LIN {X 0,Y 220.383,Z 219.803,A -85,B 0,C 180,E1 -20268.834,E2 -20268.834} C_VEL
LIN {X 0,Y 222.239,Z 208.514,A -85,B 0,C 180,E1 -20275.269,E2 -20275.269} C_VEL
LIN {X 0,Y 223.877,Z 201.722,A -85,B 0,C 180,E1 -20279.111,E2 -20279.111} C_VEL
LIN {X 0,Y 223.579,Z 198.542,A -85,B 0,C 180,E1 -20280.967,E2 -20280.967} C_VEL
LIN {X 0,Y 221.946,Z 190.437,A -85,B 0,C 180,E1 -20285.855,E2 -20285.855} C_VEL
LIN {X 0,Y 220.93,Z 184.96,A -85,B 0,C 180,E1 -20289.374,E2 -20289.374} C_VEL
LIN {X 0,Y 220.782,Z 184.985,A -85,B 0,C 180,E1 -20294.447,E2 -20294.447} C_VEL
LIN {X 0,Y 220.845,Z 184.972,A -85,B 0,C 180,E1 -20298.065,E2 -20298.065} C_VEL
LIN {X 0,Y 220.829,Z 184.976,A -85,B 0,C 180,E1 -20302.71,E2 -20302.71} C_VEL
LIN {X 0,Y 220.813,Z 184.976,A -85,B 0,C 180,E1 -20307.243,E2 -20307.243} C_VEL
LIN {X 0,Y 220.816,Z 184.978,A -85,B 0,C 180,E1 -20311.483,E2 -20311.483} C_VEL
LIN {X 0,Y 220.85,Z 184.972,A -85,B 0,C 180,E1 -20315.563,E2 -20315.563} C_VEL
LIN {X 0,Y 220.873,Z 184.973,A -85,B 0,C 180,E1 -20319.512,E2 -20319.512} C_VEL
LIN {X 0,Y 221.004,Z 184.953,A -85,B 0,C 180,E1 -20323.369,E2 -20323.369} C_VEL
LIN {X 0,Y 221.1,Z 184.943,A -85,B 0,C 180,E1 -20329.005,E2 -20329.005} C_VEL
LIN {X 0,Y 221.276,Z 184.918,A -85,B 0,C 180,E1 -20332.701,E2 -20332.701} C_VEL
LIN {X 0,Y 221.503,Z 184.891,A -85,B 0,C 180,E1 -20338.182,E2 -20338.182} C_VEL
LIN {X 0,Y 221.498,Z 184.891,A -85,B 0,C 180,E1 -20341.818,E2 -20341.818} C_VEL
LIN {X 0,Y 221.277,Z 184.918,A -85,B 0,C 180,E1 -20347.299,E2 -20347.299} C_VEL
LIN {X 0,Y 221.1,Z 184.943,A -85,B 0,C 180,E1 -20350.995,E2 -20350.995} C_VEL
LIN {X 0,Y 221.004,Z 184.953,A -85,B 0,C 180,E1 -20356.631,E2 -20356.631} C_VEL
LIN {X 0,Y 220.876,Z 184.973,A -85,B 0,C 180,E1 -20360.488,E2 -20360.488} C_VEL
LIN {X 0,Y 220.836,Z 184.974,A -85,B 0,C 180,E1 -20364.439,E2 -20364.439} C_VEL
LIN {X 0,Y 220.793,Z 184.981,A -85,B 0,C 180,E1 -20368.52,E2 -20368.52} C_VEL
LIN {X 0,Y 220.807,Z 184.977,A -85,B 0,C 180,E1 -20372.758,E2 -20372.758} C_VEL
LIN {X 0,Y 220.828,Z 184.976,A -85,B 0,C 180,E1 -20377.29,E2 -20377.29} C_VEL
LIN {X 0,Y 220.792,Z 184.979,A -85,B 0,C 180,E1 -20381.947,E2 -20381.947} C_VEL
LIN {X 0,Y 220.768,Z 184.986,A -85,B 0,C 180,E1 -20385.549,E2 -20385.549} C_VEL
LIN {X 0,Y 220.799,Z 184.978,A -85,B 0,C 180,E1 -20390.466,E2 -20390.466} C_VEL
LIN {X 0,Y 220.795,Z 184.983,A -85,B 0,C 180,E1 -20395.048,E2 -20395.048} C_VEL
LIN {X 0,Y 220.863,Z 184.969,A -85,B 0,C 180,E1 -20399.398,E2 -20399.398} C_VEL
LIN {X 0,Y 220.891,Z 184.968,A -85,B 0,C 180,E1 -20403.553,E2 -20403.553} C_VEL
LIN {X 0,Y 220.875,Z 184.968,A -85,B 0,C 180,E1 -20407.556,E2 -20407.556} C_VEL
LIN {X 0,Y 220.982,Z 184.96,A -85,B 0,C 180,E1 -20412.574,E2 -20412.574} C_VEL
LIN {X 0,Y 221.012,Z 184.95,A -85,B 0,C 180,E1 -20417.142,E2 -20417.142} C_VEL
LIN {X 0,Y 221.258,Z 184.923,A -85,B 0,C 180,E1 -20420.865,E2 -20420.865} C_VEL
LIN {X 0,Y 221.312,Z 184.916,A -85,B 0,C 180,E1 -20422.705,E2 -20422.705} C_VEL
LIN {X 0,Y 221.511,Z 184.894,A -85,B 0,C 180,E1 -20428.185,E2 -20428.185} C_VEL
LIN {X 0,Y 221.51,Z 184.894,A -85,B 0,C 180,E1 -20431.821,E2 -20431.821} C_VEL
LIN {X 0,Y 221.314,Z 184.916,A -85,B 0,C 180,E1 -20437.3,E2 -20437.3} C_VEL
LIN {X 0,Y 221.115,Z 184.94,A -85,B 0,C 180,E1 -20440.997,E2 -20440.997} C_VEL
LIN {X 0,Y 221.02,Z 184.952,A -85,B 0,C 180,E1 -20446.632,E2 -20446.632} C_VEL
LIN {X 0,Y 220.886,Z 184.967,A -85,B 0,C 180,E1 -20450.49,E2 -20450.49} C_VEL
LIN {X 0,Y 220.803,Z 184.979,A -85,B 0,C 180,E1 -20454.445,E2 -20454.445} C_VEL
LIN {X 0,Y 220.804,Z 184.979,A -85,B 0,C 180,E1 -20458.521,E2 -20458.521} C_VEL
LIN {X 0,Y 220.818,Z 184.979,A -85,B 0,C 180,E1 -20462.759,E2 -20462.759} C_VEL
LIN {X 0,Y 220.815,Z 184.976,A -85,B 0,C 180,E1 -20467.28,E2 -20467.28} C_VEL
LIN {X 0,Y 220.758,Z 184.985,A -85,B 0,C 180,E1 -20471.959,E2 -20471.959} C_VEL
LIN {X 0,Y 220.776,Z 184.981,A -85,B 0,C 180,E1 -20475.547,E2 -20475.547} C_VEL
LIN {X 0,Y 220.818,Z 184.98,A -85,B 0,C 180,E1 -20480.465,E2 -20480.465} C_VEL
LIN {X 0,Y 221.099,Z 185.049,A -85,B 0,C 180,E1 -20484.682,E2 -20484.682} C_VEL
LIN {X 0,Y 221.776,Z 188.632,A -85,B 0,C 180,E1 -20487.403,E2 -20487.403} C_VEL
LIN {X 0,Y 221.812,Z 191.54,A -85,B 0,C 180,E1 -20489.539,E2 -20489.539} C_VEL
LIN {X 0,Y 220.785,Z 198.517,A -85,B 0,C 180,E1 -20494.55,E2 -20494.55} C_VEL
LIN {X 0,Y 219.989,Z 205.404,A -85,B 0,C 180,E1 -20499.426,E2 -20499.426} C_VEL
LIN {X 0,Y 219.304,Z 213.531,A -85,B 0,C 180,E1 -20505.145,E2 -20505.145} C_VEL
LIN {X 0,Y 219.238,Z 217.231,A -85,B 0,C 180,E1 -20507.739,E2 -20507.739} C_VEL
LIN {X 0,Y 219.799,Z 228.527,A -85,B 0,C 180,E1 -20508.939,E2 -20508.939} C_VEL
LIN {X 0,Y 220.545,Z 237.591,A -85,B 0,C 180,E1 -20510.138,E2 -20510.138} C_VEL
LIN {X 0,Y 220.063,Z 248.605,A -85,B 0,C 180,E1 -20511.998,E2 -20511.998} C_VEL
LIN {X 0,Y 219.533,Z 258.766,A -85,B 0,C 180,E1 -20514.185,E2 -20514.185} C_VEL
LIN {X 0,Y 219.318,Z 266.733,A -85,B 0,C 180,E1 -20516.326,E2 -20516.326} C_VEL
LIN {X 0,Y 218.971,Z 273.609,A -85,B 0,C 180,E1 -20518.621,E2 -20518.621} C_VEL
LIN {X 0,Y 218.926,Z 279.136,A -85,B 0,C 180,E1 -20520.92,E2 -20520.92} C_VEL
LIN {X 0,Y 219.375,Z 284.347,A -85,B 0,C 180,E1 -20523.674,E2 -20523.674} C_VEL
LIN {X 0,Y 220.373,Z 288.134,A -85,B 0,C 180,E1 -20526.409,E2 -20526.409} C_VEL
LIN {X 0,Y 221.649,Z 290.652,A -85,B 0,C 180,E1 -20529.122,E2 -20529.122} C_VEL
LIN {X 0,Y 222.867,Z 291.672,A -85,B 0,C 180,E1 -20530.907,E2 -20530.907} C_VEL
LIN {X 0,Y 224.323,Z 292.16,A -85,B 0,C 180,E1 -20532.669,E2 -20532.669} C_VEL
LIN {X 0,Y 226.248,Z 292.142,A -85,B 0,C 180,E1 -20534.389,E2 -20534.389} C_VEL
LIN {X 0,Y 228.21,Z 291.601,A -85,B 0,C 180,E1 -20536.091,E2 -20536.091} C_VEL
LIN {X 0,Y 230.547,Z 290.562,A -85,B 0,C 180,E1 -20537.749,E2 -20537.749} C_VEL
LIN {X 0,Y 234.632,Z 287.997,A -85,B 0,C 180,E1 -20540.149,E2 -20540.149} C_VEL
LIN {X 0,Y 239.086,Z 284.255,A -85,B 0,C 180,E1 -20542.466,E2 -20542.466} C_VEL
LIN {X 0,Y 242.31,Z 281.065,A -85,B 0,C 180,E1 -20543.958,E2 -20543.958} C_VEL
LIN {X 0,Y 243.63,Z 279.399,A -85,B 0,C 180,E1 -20544.726,E2 -20544.726} C_VEL
LIN {X 0,Y 246.198,Z 274.482,A -85,B 0,C 180,E1 -20547.177,E2 -20547.177} C_VEL
LIN {X 0,Y 248.143,Z 269.374,A -85,B 0,C 180,E1 -20549.712,E2 -20549.712} C_VEL
LIN {X 0,Y 250.03,Z 263.054,A -85,B 0,C 180,E1 -20553.028,E2 -20553.028} C_VEL
LIN {X 0,Y 250.761,Z 259.802,A -85,B 0,C 180,E1 -20555.088,E2 -20555.088} C_VEL
LIN {X 0,Y 250.91,Z 258.67,A -85,B 0,C 180,E1 -20556.03,E2 -20556.03} C_VEL
LIN {X 0,Y 251.075,Z 256.645,A -85,B 0,C 180,E1 -20558.39,E2 -20558.39} C_VEL
LIN {X 0,Y 251.135,Z 255.646,A -85,B 0,C 180,E1 -20560.92,E2 -20560.92} C_VEL
LIN {X 0,Y 251.591,Z 255.794,A -85,B 0,C 180,E1 -20564.296,E2 -20564.296} C_VEL
LIN {X 0,Y 252.211,Z 256.685,A -85,B 0,C 180,E1 -20566.428,E2 -20566.428} C_VEL
LIN {X 0,Y 252.859,Z 258.56,A -85,B 0,C 180,E1 -20568.629,E2 -20568.629} C_VEL
LIN {X 0,Y 253.665,Z 261.185,A -85,B 0,C 180,E1 -20570.875,E2 -20570.875} C_VEL
LIN {X 0,Y 254.443,Z 264.949,A -85,B 0,C 180,E1 -20573.227,E2 -20573.227} C_VEL
LIN {X 0,Y 254.346,Z 266.588,A -85,B 0,C 180,E1 -20573.944,E2 -20573.944} C_VEL
LIN {X 0,Y 251.506,Z 274.816,A -85,B 0,C 180,E1 -20576.501,E2 -20576.501} C_VEL
LIN {X 0,Y 250.329,Z 277.426,A -85,B 0,C 180,E1 -20577.284,E2 -20577.284} C_VEL
LIN {X 0,Y 246.162,Z 283.563,A -85,B 0,C 180,E1 -20578.844,E2 -20578.844} C_VEL
LIN {X 0,Y 243.112,Z 287.073,A -85,B 0,C 180,E1 -20579.71,E2 -20579.71} C_VEL
LIN {X 0,Y 236.799,Z 292.522,A -85,B 0,C 180,E1 -20580.998,E2 -20580.998} C_VEL
LIN {X 0,Y 230.529,Z 297.239,A -85,B 0,C 180,E1 -20582.454,E2 -20582.454} C_VEL
LIN {X 0,Y 227.594,Z 299.611,A -85,B 0,C 180,E1 -20583.576,E2 -20583.576} C_VEL
LIN {X 0,Y 223.623,Z 303.227,A -85,B 0,C 180,E1 -20585.883,E2 -20585.883} C_VEL
LIN {X 0,Y 219.258,Z 306.967,A -85,B 0,C 180,E1 -20589.351,E2 -20589.351} C_VEL
LIN {X 0,Y 215.694,Z 309.301,A -85,B 0,C 180,E1 -20592.945,E2 -20592.945} C_VEL
LIN {X 0,Y 213.363,Z 310.182,A -85,B 0,C 180,E1 -20596.666,E2 -20596.666} C_VEL
LIN {X 0,Y 212.177,Z 309.707,A -85,B 0,C 180,E1 -20600.464,E2 -20600.464} C_VEL
LIN {X 0,Y 212.07,Z 307.767,A -85,B 0,C 180,E1 -20604.291,E2 -20604.291} C_VEL
LIN {X 0,Y 212.215,Z 306.227,A -85,B 0,C 180,E1 -20606.199,E2 -20606.199} C_VEL
LIN {X 0,Y 212.782,Z 303.097,A -85,B 0,C 180,E1 -20609.051,E2 -20609.051} C_VEL
LIN {X 0,Y 213.004,Z 300.337,A -85,B 0,C 180,E1 -20610.942,E2 -20610.942} C_VEL
LIN {X 0,Y 213.038,Z 295.011,A -85,B 0,C 180,E1 -20613.78,E2 -20613.78} C_VEL
LIN {X 0,Y 213.16,Z 288.15,A -85,B 0,C 180,E1 -20616.623,E2 -20616.623} C_VEL
LIN {X 0,Y 213.282,Z 279.264,A -85,B 0,C 180,E1 -20619.48,E2 -20619.48} C_VEL
LIN {X 0,Y 213.737,Z 269.98,A -85,B 0,C 180,E1 -20621.856,E2 -20621.856} C_VEL
LIN {X 0,Y 214.337,Z 259.585,A -85,B 0,C 180,E1 -20623.991,E2 -20623.991} C_VEL
LIN {X 0,Y 215.12,Z 247.855,A -85,B 0,C 180,E1 -20625.876,E2 -20625.876} C_VEL
LIN {X 0,Y 214.061,Z 235.879,A -85,B 0,C 180,E1 -20627.3,E2 -20627.3} C_VEL
LIN {X 0,Y 213.328,Z 223.422,A -85,B 0,C 180,E1 -20628.407,E2 -20628.407} C_VEL
LIN {X 0,Y 213.308,Z 219.864,A -85,B 0,C 180,E1 -20628.683,E2 -20628.683} C_VEL
LIN {X 0,Y 215.064,Z 208.981,A -85,B 0,C 180,E1 -20635.136,E2 -20635.136} C_VEL
LIN {X 0,Y 216.744,Z 202.237,A -85,B 0,C 180,E1 -20639.099,E2 -20639.099} C_VEL
LIN {X 0,Y 216.769,Z 200.445,A -85,B 0,C 180,E1 -20640.164,E2 -20640.164} C_VEL
LIN {X 0,Y 215.08,Z 192.314,A -85,B 0,C 180,E1 -20645.223,E2 -20645.223} C_VEL
LIN {X 0,Y 213.891,Z 185.837,A -85,B 0,C 180,E1 -20649.383,E2 -20649.383} C_VEL
LIN {X 0,Y 213.74,Z 185.859,A -85,B 0,C 180,E1 -20653.665,E2 -20653.665} C_VEL
LIN {X 0,Y 213.804,Z 185.851,A -85,B 0,C 180,E1 -20656.346,E2 -20656.346} C_VEL
LIN {X 0,Y 213.786,Z 185.852,A -85,B 0,C 180,E1 -20659.116,E2 -20659.116} C_VEL
LIN {X 0,Y 213.745,Z 185.859,A -85,B 0,C 180,E1 -20663.712,E2 -20663.712} C_VEL
LIN {X 0,Y 213.76,Z 185.859,A -85,B 0,C 180,E1 -20668.261,E2 -20668.261} C_VEL
LIN {X 0,Y 213.815,Z 185.848,A -85,B 0,C 180,E1 -20672.601,E2 -20672.601} C_VEL
LIN {X 0,Y 213.808,Z 185.85,A -85,B 0,C 180,E1 -20676.972,E2 -20676.972} C_VEL
LIN {X 0,Y 213.932,Z 185.832,A -85,B 0,C 180,E1 -20682.802,E2 -20682.802} C_VEL
LIN {X 0,Y 213.968,Z 185.831,A -85,B 0,C 180,E1 -20686.707,E2 -20686.707} C_VEL
LIN {X 0,Y 214.155,Z 185.805,A -85,B 0,C 180,E1 -20690.556,E2 -20690.556} C_VEL
LIN {X 0,Y 214.214,Z 185.797,A -85,B 0,C 180,E1 -20692.459,E2 -20692.459} C_VEL
LIN {X 0,Y 214.436,Z 185.771,A -85,B 0,C 180,E1 -20698.122,E2 -20698.122} C_VEL
LIN {X 0,Y 214.537,Z 185.756,A -85,B 0,C 180,E1 -20700,E2 -20700} C_VEL
LIN {X 0,Y 214.431,Z 185.772,A -85,B 0,C 180,E1 -20701.878,E2 -20701.878} C_VEL
LIN {X 0,Y 214.215,Z 185.797,A -85,B 0,C 180,E1 -20707.541,E2 -20707.541} C_VEL
LIN {X 0,Y 214.032,Z 185.822,A -85,B 0,C 180,E1 -20711.362,E2 -20711.362} C_VEL
LIN {X 0,Y 213.921,Z 185.835,A -85,B 0,C 180,E1 -20715.238,E2 -20715.238} C_VEL
LIN {X 0,Y 213.825,Z 185.848,A -85,B 0,C 180,E1 -20719.189,E2 -20719.189} C_VEL
LIN {X 0,Y 213.791,Z 185.852,A -85,B 0,C 180,E1 -20723.233,E2 -20723.233} C_VEL
LIN {X 0,Y 213.775,Z 185.853,A -85,B 0,C 180,E1 -20727.43,E2 -20727.43} C_VEL
LIN {X 0,Y 213.75,Z 185.86,A -85,B 0,C 180,E1 -20731.74,E2 -20731.74} C_VEL
LIN {X 0,Y 213.742,Z 185.859,A -85,B 0,C 180,E1 -20736.289,E2 -20736.289} C_VEL
LIN {X 0,Y 213.723,Z 185.861,A -85,B 0,C 180,E1 -20741.123,E2 -20741.123} C_VEL
LIN {X 0,Y 213.739,Z 185.859,A -85,B 0,C 180,E1 -20743.67,E2 -20743.67} C_VEL
LIN {X 0,Y 213.704,Z 185.864,A -85,B 0,C 180,E1 -20748.878,E2 -20748.878} C_VEL
LIN {X 0,Y 213.737,Z 185.86,A -85,B 0,C 180,E1 -20753.715,E2 -20753.715} C_VEL
LIN {X 0,Y 213.789,Z 185.853,A -85,B 0,C 180,E1 -20758.728,E2 -20758.728} C_VEL
LIN {X 0,Y 213.821,Z 185.849,A -85,B 0,C 180,E1 -20762.606,E2 -20762.606} C_VEL
LIN {X 0,Y 213.848,Z 185.845,A -85,B 0,C 180,E1 -20766.956,E2 -20766.956} C_VEL
LIN {X 0,Y 213.93,Z 185.837,A -85,B 0,C 180,E1 -20772.308,E2 -20772.308} C_VEL
LIN {X 0,Y 213.953,Z 185.831,A -85,B 0,C 180,E1 -20776.71,E2 -20776.71} C_VEL
LIN {X 0,Y 214.196,Z 185.804,A -85,B 0,C 180,E1 -20780.561,E2 -20780.561} C_VEL
LIN {X 0,Y 214.248,Z 185.797,A -85,B 0,C 180,E1 -20782.463,E2 -20782.463} C_VEL
LIN {X 0,Y 214.445,Z 185.774,A -85,B 0,C 180,E1 -20788.125,E2 -20788.125} C_VEL
LIN {X 0,Y 214.444,Z 185.774,A -85,B 0,C 180,E1 -20791.881,E2 -20791.881} C_VEL
LIN {X 0,Y 214.251,Z 185.797,A -85,B 0,C 180,E1 -20797.542,E2 -20797.542} C_VEL
LIN {X 0,Y 214.046,Z 185.822,A -85,B 0,C 180,E1 -20801.365,E2 -20801.365} C_VEL
LIN {X 0,Y 213.938,Z 185.835,A -85,B 0,C 180,E1 -20805.239,E2 -20805.239} C_VEL
LIN {X 0,Y 213.838,Z 185.849,A -85,B 0,C 180,E1 -20809.19,E2 -20809.19} C_VEL
LIN {X 0,Y 213.788,Z 185.854,A -85,B 0,C 180,E1 -20813.237,E2 -20813.237} C_VEL
LIN {X 0,Y 213.789,Z 185.853,A -85,B 0,C 180,E1 -20817.429,E2 -20817.429} C_VEL
LIN {X 0,Y 213.764,Z 185.855,A -85,B 0,C 180,E1 -20821.741,E2 -20821.741} C_VEL
LIN {X 0,Y 213.75,Z 185.858,A -85,B 0,C 180,E1 -20826.29,E2 -20826.29} C_VEL
LIN {X 0,Y 213.705,Z 185.864,A -85,B 0,C 180,E1 -20831.13,E2 -20831.13} C_VEL
LIN {X 0,Y 213.709,Z 185.863,A -85,B 0,C 180,E1 -20833.681,E2 -20833.681} C_VEL
LIN {X 0,Y 213.711,Z 185.863,A -85,B 0,C 180,E1 -20836.346,E2 -20836.346} C_VEL
LIN {X 0,Y 213.791,Z 185.853,A -85,B 0,C 180,E1 -20841.348,E2 -20841.348} C_VEL
LIN {X 0,Y 214.063,Z 185.926,A -85,B 0,C 180,E1 -20844.714,E2 -20844.714} C_VEL
LIN {X 0,Y 214.817,Z 190.504,A -85,B 0,C 180,E1 -20848.284,E2 -20848.284} C_VEL
LIN {X 0,Y 214.282,Z 194.938,A -85,B 0,C 180,E1 -20851.583,E2 -20851.583} C_VEL
LIN {X 0,Y 213.301,Z 201.913,A -85,B 0,C 180,E1 -20856.71,E2 -20856.71} C_VEL
LIN {X 0,Y 212.547,Z 208.755,A -85,B 0,C 180,E1 -20861.692,E2 -20861.692} C_VEL
LIN {X 0,Y 212.122,Z 215.525,A -85,B 0,C 180,E1 -20866.59,E2 -20866.59} C_VEL
LIN {X 0,Y 212.156,Z 217.294,A -85,B 0,C 180,E1 -20867.869,E2 -20867.869} C_VEL
LIN {X 0,Y 212.885,Z 229.982,A -85,B 0,C 180,E1 -20869.298,E2 -20869.298} C_VEL
LIN {X 0,Y 213.44,Z 238.744,A -85,B 0,C 180,E1 -20870.524,E2 -20870.524} C_VEL
LIN {X 0,Y 212.968,Z 249.317,A -85,B 0,C 180,E1 -20872.415,E2 -20872.415} C_VEL
LIN {X 0,Y 212.521,Z 257.854,A -85,B 0,C 180,E1 -20874.307,E2 -20874.307} C_VEL
LIN {X 0,Y 212.274,Z 266.55,A -85,B 0,C 180,E1 -20876.679,E2 -20876.679} C_VEL
LIN {X 0,Y 211.927,Z 274.714,A -85,B 0,C 180,E1 -20879.525,E2 -20879.525} C_VEL
LIN {X 0,Y 211.986,Z 280.073,A -85,B 0,C 180,E1 -20881.9,E2 -20881.9} C_VEL
LIN {X 0,Y 212.598,Z 285.136,A -85,B 0,C 180,E1 -20884.741,E2 -20884.741} C_VEL
LIN {X 0,Y 213.806,Z 288.841,A -85,B 0,C 180,E1 -20887.556,E2 -20887.556} C_VEL
LIN {X 0,Y 214.653,Z 290.584,A -85,B 0,C 180,E1 -20889.422,E2 -20889.422} C_VEL
LIN {X 0,Y 215.911,Z 291.844,A -85,B 0,C 180,E1 -20891.263,E2 -20891.263} C_VEL
LIN {X 0,Y 217.433,Z 292.568,A -85,B 0,C 180,E1 -20893.077,E2 -20893.077} C_VEL
LIN {X 0,Y 219.401,Z 292.78,A -85,B 0,C 180,E1 -20894.849,E2 -20894.849} C_VEL
LIN {X 0,Y 221.463,Z 292.511,A -85,B 0,C 180,E1 -20896.595,E2 -20896.595} C_VEL
LIN {X 0,Y 223.875,Z 291.714,A -85,B 0,C 180,E1 -20898.296,E2 -20898.296} C_VEL
LIN {X 0,Y 226.647,Z 290.42,A -85,B 0,C 180,E1 -20899.944,E2 -20899.944} C_VEL
LIN {X 0,Y 231.135,Z 287.501,A -85,B 0,C 180,E1 -20902.339,E2 -20902.339} C_VEL
LIN {X 0,Y 236.095,Z 283.421,A -85,B 0,C 180,E1 -20904.63,E2 -20904.63} C_VEL
LIN {X 0,Y 237.579,Z 281.888,A -85,B 0,C 180,E1 -20905.4,E2 -20905.4} C_VEL
LIN {X 0,Y 240.458,Z 277.435,A -85,B 0,C 180,E1 -20907.882,E2 -20907.882} C_VEL
LIN {X 0,Y 242.733,Z 272.796,A -85,B 0,C 180,E1 -20910.444,E2 -20910.444} C_VEL
LIN {X 0,Y 245.023,Z 267.195,A -85,B 0,C 180,E1 -20913.711,E2 -20913.711} C_VEL
LIN {X 0,Y 246.057,Z 264.079,A -85,B 0,C 180,E1 -20915.974,E2 -20915.974} C_VEL
LIN {X 0,Y 246.476,Z 261.855,A -85,B 0,C 180,E1 -20918.852,E2 -20918.852} C_VEL
LIN {X 0,Y 246.672,Z 261.171,A -85,B 0,C 180,E1 -20920.943,E2 -20920.943} C_VEL
LIN {X 0,Y 246.926,Z 261.137,A -85,B 0,C 180,E1 -20923.086,E2 -20923.086} C_VEL
LIN {X 0,Y 247.401,Z 261.685,A -85,B 0,C 180,E1 -20925.25,E2 -20925.25} C_VEL
LIN {X 0,Y 247.945,Z 263.026,A -85,B 0,C 180,E1 -20927.474,E2 -20927.474} C_VEL
LIN {X 0,Y 248.585,Z 265.172,A -85,B 0,C 180,E1 -20929.76,E2 -20929.76} C_VEL
LIN {X 0,Y 249.153,Z 268.435,A -85,B 0,C 180,E1 -20932.168,E2 -20932.168} C_VEL
LIN {X 0,Y 249.169,Z 270.29,A -85,B 0,C 180,E1 -20933.2,E2 -20933.2} C_VEL
LIN {X 0,Y 246.665,Z 276.32,A -85,B 0,C 180,E1 -20935.258,E2 -20935.258} C_VEL
LIN {X 0,Y 245.111,Z 279.384,A -85,B 0,C 180,E1 -20936.255,E2 -20936.255} C_VEL
LIN {X 0,Y 238.884,Z 287.459,A -85,B 0,C 180,E1 -20938.517,E2 -20938.517} C_VEL
LIN {X 0,Y 232.634,Z 294.496,A -85,B 0,C 180,E1 -20941.092,E2 -20941.092} C_VEL
LIN {X 0,Y 227.594,Z 299.611,A -85,B 0,C 180,E1 -20943.576,E2 -20943.576} C_VEL
LIN {X 0,Y 224.729,Z 301.802,A -85,B 0,C 180,E1 -20944.777,E2 -20944.777} C_VEL
LIN {X 0,Y 218.799,Z 304.886,A -85,B 0,C 180,E1 -20946.677,E2 -20946.677} C_VEL
LIN {X 0,Y 213.226,Z 307.124,A -85,B 0,C 180,E1 -20948.742,E2 -20948.742} C_VEL
LIN {X 0,Y 210.967,Z 308.051,A -85,B 0,C 180,E1 -20950.177,E2 -20950.177} C_VEL
LIN {X 0,Y 208.917,Z 309.041,A -85,B 0,C 180,E1 -20952.373,E2 -20952.373} C_VEL
LIN {X 0,Y 207.468,Z 309.495,A -85,B 0,C 180,E1 -20954.273,E2 -20954.273} C_VEL
LIN {X 0,Y 205.699,Z 309.337,A -85,B 0,C 180,E1 -20958.168,E2 -20958.168} C_VEL
LIN {X 0,Y 205,Z 307.828,A -85,B 0,C 180,E1 -20962.115,E2 -20962.115} C_VEL
LIN {X 0,Y 205.087,Z 306.522,A -85,B 0,C 180,E1 -20964.096,E2 -20964.096} C_VEL
LIN {X 0,Y 205.714,Z 302.691,A -85,B 0,C 180,E1 -20968.039,E2 -20968.039} C_VEL
LIN {X 0,Y 206.06,Z 300.058,A -85,B 0,C 180,E1 -20969.997,E2 -20969.997} C_VEL
LIN {X 0,Y 206.137,Z 294.882,A -85,B 0,C 180,E1 -20972.928,E2 -20972.928} C_VEL
LIN {X 0,Y 206.229,Z 288.195,A -85,B 0,C 180,E1 -20975.865,E2 -20975.865} C_VEL
LIN {X 0,Y 206.274,Z 280.962,A -85,B 0,C 180,E1 -20978.373,E2 -20978.373} C_VEL
LIN {X 0,Y 206.635,Z 272.437,A -85,B 0,C 180,E1 -20980.778,E2 -20980.778} C_VEL
LIN {X 0,Y 207.143,Z 262.818,A -85,B 0,C 180,E1 -20982.986,E2 -20982.986} C_VEL
LIN {X 0,Y 207.862,Z 250.619,A -85,B 0,C 180,E1 -20985.187,E2 -20985.187} C_VEL
LIN {X 0,Y 207.974,Z 245.538,A -85,B 0,C 180,E1 -20985.933,E2 -20985.933} C_VEL
LIN {X 0,Y 206.781,Z 232.916,A -85,B 0,C 180,E1 -20987.404,E2 -20987.404} C_VEL
LIN {X 0,Y 206.262,Z 220.901,A -85,B 0,C 180,E1 -20988.432,E2 -20988.432} C_VEL
LIN {X 0,Y 206.223,Z 219.776,A -85,B 0,C 180,E1 -20988.565,E2 -20988.565} C_VEL
LIN {X 0,Y 208.27,Z 207.727,A -85,B 0,C 180,E1 -20996.016,E2 -20996.016} C_VEL
LIN {X 0,Y 209.665,Z 202.24,A -85,B 0,C 180,E1 -20999.363,E2 -20999.363} C_VEL
LIN {X 0,Y 209.269,Z 199.049,A -85,B 0,C 180,E1 -21001.365,E2 -21001.365} C_VEL
LIN {X 0,Y 207.854,Z 192.27,A -85,B 0,C 180,E1 -21005.757,E2 -21005.757} C_VEL
LIN {X 0,Y 206.826,Z 186.717,A -85,B 0,C 180,E1 -21009.578,E2 -21009.578} C_VEL
LIN {X 0,Y 206.7,Z 186.734,A -85,B 0,C 180,E1 -21015.558,E2 -21015.558} C_VEL
LIN {X 0,Y 206.716,Z 186.734,A -85,B 0,C 180,E1 -21019.761,E2 -21019.761} C_VEL
LIN {X 0,Y 206.716,Z 186.737,A -85,B 0,C 180,E1 -21022.268,E2 -21022.268} C_VEL
LIN {X 0,Y 206.696,Z 186.734,A -85,B 0,C 180,E1 -21027.042,E2 -21027.042} C_VEL
LIN {X 0,Y 206.754,Z 186.73,A -85,B 0,C 180,E1 -21032.096,E2 -21032.096} C_VEL
LIN {X 0,Y 206.743,Z 186.73,A -85,B 0,C 180,E1 -21036.602,E2 -21036.602} C_VEL
LIN {X 0,Y 206.861,Z 186.713,A -85,B 0,C 180,E1 -21042.195,E2 -21042.195} C_VEL
LIN {X 0,Y 206.902,Z 186.711,A -85,B 0,C 180,E1 -21046.245,E2 -21046.245} C_VEL
LIN {X 0,Y 207.093,Z 186.685,A -85,B 0,C 180,E1 -21050.23,E2 -21050.23} C_VEL
LIN {X 0,Y 207.061,Z 186.69,A -85,B 0,C 180,E1 -21054.156,E2 -21054.156} C_VEL
LIN {X 0,Y 207.373,Z 186.651,A -85,B 0,C 180,E1 -21058.058,E2 -21058.058} C_VEL
LIN {X 0,Y 207.502,Z 186.632,A -85,B 0,C 180,E1 -21060,E2 -21060} C_VEL
LIN {X 0,Y 207.368,Z 186.651,A -85,B 0,C 180,E1 -21061.942,E2 -21061.942} C_VEL
LIN {X 0,Y 207.155,Z 186.676,A -85,B 0,C 180,E1 -21067.799,E2 -21067.799} C_VEL
LIN {X 0,Y 206.969,Z 186.702,A -85,B 0,C 180,E1 -21071.756,E2 -21071.756} C_VEL
LIN {X 0,Y 206.855,Z 186.715,A -85,B 0,C 180,E1 -21075.772,E2 -21075.772} C_VEL
LIN {X 0,Y 206.768,Z 186.727,A -85,B 0,C 180,E1 -21079.871,E2 -21079.871} C_VEL
LIN {X 0,Y 206.727,Z 186.734,A -85,B 0,C 180,E1 -21084.077,E2 -21084.077} C_VEL
LIN {X 0,Y 206.677,Z 186.74,A -85,B 0,C 180,E1 -21088.429,E2 -21088.429} C_VEL
LIN {X 0,Y 206.691,Z 186.735,A -85,B 0,C 180,E1 -21092.959,E2 -21092.959} C_VEL
LIN {X 0,Y 206.712,Z 186.732,A -85,B 0,C 180,E1 -21095.322,E2 -21095.322} C_VEL
LIN {X 0,Y 206.665,Z 186.74,A -85,B 0,C 180,E1 -21100.25,E2 -21100.25} C_VEL
LIN {X 0,Y 206.651,Z 186.74,A -85,B 0,C 180,E1 -21104.428,E2 -21104.428} C_VEL
LIN {X 0,Y 206.653,Z 186.741,A -85,B 0,C 180,E1 -21109.752,E2 -21109.752} C_VEL
LIN {X 0,Y 206.692,Z 186.737,A -85,B 0,C 180,E1 -21114.692,E2 -21114.692} C_VEL
LIN {X 0,Y 206.717,Z 186.731,A -85,B 0,C 180,E1 -21119.342,E2 -21119.342} C_VEL
LIN {X 0,Y 206.729,Z 186.732,A -85,B 0,C 180,E1 -21123.775,E2 -21123.775} C_VEL
LIN {X 0,Y 206.754,Z 186.727,A -85,B 0,C 180,E1 -21128.047,E2 -21128.047} C_VEL
LIN {X 0,Y 206.874,Z 186.715,A -85,B 0,C 180,E1 -21132.2,E2 -21132.2} C_VEL
LIN {X 0,Y 206.895,Z 186.712,A -85,B 0,C 180,E1 -21136.248,E2 -21136.248} C_VEL
LIN {X 0,Y 207.132,Z 186.684,A -85,B 0,C 180,E1 -21140.236,E2 -21140.236} C_VEL
LIN {X 0,Y 207.189,Z 186.678,A -85,B 0,C 180,E1 -21142.205,E2 -21142.205} C_VEL
LIN {X 0,Y 207.382,Z 186.653,A -85,B 0,C 180,E1 -21148.061,E2 -21148.061} C_VEL
LIN {X 0,Y 207.484,Z 186.642,A -85,B 0,C 180,E1 -21150.003,E2 -21150.003} C_VEL
LIN {X 0,Y 207.381,Z 186.653,A -85,B 0,C 180,E1 -21151.945,E2 -21151.945} C_VEL
LIN {X 0,Y 207.192,Z 186.678,A -85,B 0,C 180,E1 -21157.801,E2 -21157.801} C_VEL
LIN {X 0,Y 206.979,Z 186.7,A -85,B 0,C 180,E1 -21161.758,E2 -21161.758} C_VEL
LIN {X 0,Y 206.871,Z 186.716,A -85,B 0,C 180,E1 -21165.773,E2 -21165.773} C_VEL
LIN {X 0,Y 206.764,Z 186.726,A -85,B 0,C 180,E1 -21169.874,E2 -21169.874} C_VEL
LIN {X 0,Y 206.705,Z 186.735,A -85,B 0,C 180,E1 -21174.082,E2 -21174.082} C_VEL
LIN {X 0,Y 206.692,Z 186.736,A -85,B 0,C 180,E1 -21178.43,E2 -21178.43} C_VEL
LIN {X 0,Y 206.701,Z 186.739,A -85,B 0,C 180,E1 -21182.96,E2 -21182.96} C_VEL
LIN {X 0,Y 206.679,Z 186.736,A -85,B 0,C 180,E1 -21187.743,E2 -21187.743} C_VEL
LIN {X 0,Y 206.638,Z 186.743,A -85,B 0,C 180,E1 -21191.561,E2 -21191.561} C_VEL
LIN {X 0,Y 206.638,Z 186.742,A -85,B 0,C 180,E1 -21195.584,E2 -21195.584} C_VEL
LIN {X 0,Y 206.684,Z 186.738,A -85,B 0,C 180,E1 -21199.754,E2 -21199.754} C_VEL
LIN {X 0,Y 207.033,Z 186.775,A -85,B 0,C 180,E1 -21204.754,E2 -21204.754} C_VEL
LIN {X 0,Y 207.692,Z 190.556,A -85,B 0,C 180,E1 -21207.78,E2 -21207.78} C_VEL
LIN {X 0,Y 207.404,Z 194.166,A -85,B 0,C 180,E1 -21210.571,E2 -21210.571} C_VEL
LIN {X 0,Y 206.359,Z 201.149,A -85,B 0,C 180,E1 -21215.878,E2 -21215.878} C_VEL
LIN {X 0,Y 205.533,Z 208.004,A -85,B 0,C 180,E1 -21221.044,E2 -21221.044} C_VEL
LIN {X 0,Y 205.051,Z 214.791,A -85,B 0,C 180,E1 -21226.118,E2 -21226.118} C_VEL
LIN {X 0,Y 205.117,Z 217.4,A -85,B 0,C 180,E1 -21228.074,E2 -21228.074} C_VEL
LIN {X 0,Y 205.754,Z 229.252,A -85,B 0,C 180,E1 -21229.421,E2 -21229.421} C_VEL
LIN {X 0,Y 206.395,Z 238.465,A -85,B 0,C 180,E1 -21230.741,E2 -21230.741} C_VEL
LIN {X 0,Y 205.949,Z 248.717,A -85,B 0,C 180,E1 -21232.611,E2 -21232.611} C_VEL
LIN {X 0,Y 205.466,Z 259.399,A -85,B 0,C 180,E1 -21235.095,E2 -21235.095} C_VEL
LIN {X 0,Y 205.234,Z 266.261,A -85,B 0,C 180,E1 -21237.056,E2 -21237.056} C_VEL
LIN {X 0,Y 204.908,Z 274.514,A -85,B 0,C 180,E1 -21240,E2 -21240} C_VEL
LIN {X 0,Y 205.115,Z 280.942,A -85,B 0,C 180,E1 -21242.946,E2 -21242.946} C_VEL
LIN {X 0,Y 205.907,Z 285.873,A -85,B 0,C 180,E1 -21245.877,E2 -21245.877} C_VEL
LIN {X 0,Y 206.795,Z 288.435,A -85,B 0,C 180,E1 -21247.813,E2 -21247.813} C_VEL
LIN {X 0,Y 207.665,Z 290.411,A -85,B 0,C 180,E1 -21249.742,E2 -21249.742} C_VEL
LIN {X 0,Y 208.966,Z 291.882,A -85,B 0,C 180,E1 -21251.642,E2 -21251.642} C_VEL
LIN {X 0,Y 210.557,Z 292.867,A -85,B 0,C 180,E1 -21253.512,E2 -21253.512} C_VEL
LIN {X 0,Y 212.562,Z 293.313,A -85,B 0,C 180,E1 -21255.338,E2 -21255.338} C_VEL
LIN {X 0,Y 214.734,Z 293.3,A -85,B 0,C 180,E1 -21257.131,E2 -21257.131} C_VEL
LIN {X 0,Y 217.224,Z 292.763,A -85,B 0,C 180,E1 -21258.877,E2 -21258.877} C_VEL
LIN {X 0,Y 220.068,Z 291.737,A -85,B 0,C 180,E1 -21260.567,E2 -21260.567} C_VEL
LIN {X 0,Y 224.731,Z 289.268,A -85,B 0,C 180,E1 -21263.011,E2 -21263.011} C_VEL
LIN {X 0,Y 229.88,Z 285.663,A -85,B 0,C 180,E1 -21265.342,E2 -21265.342} C_VEL
LIN {X 0,Y 231.5,Z 284.265,A -85,B 0,C 180,E1 -21266.117,E2 -21266.117} C_VEL
LIN {X 0,Y 233.762,Z 281.58,A -85,B 0,C 180,E1 -21267.775,E2 -21267.775} C_VEL
LIN {X 0,Y 236.699,Z 277.116,A -85,B 0,C 180,E1 -21270.56,E2 -21270.56} C_VEL
LIN {X 0,Y 239.523,Z 271.973,A -85,B 0,C 180,E1 -21273.883,E2 -21273.883} C_VEL
LIN {X 0,Y 240.711,Z 269.524,A -85,B 0,C 180,E1 -21275.728,E2 -21275.728} C_VEL
LIN {X 0,Y 241.395,Z 267.533,A -85,B 0,C 180,E1 -21278.176,E2 -21278.176} C_VEL
LIN {X 0,Y 241.751,Z 266.713,A -85,B 0,C 180,E1 -21279.76,E2 -21279.76} C_VEL
LIN {X 0,Y 241.996,Z 266.365,A -85,B 0,C 180,E1 -21281.91,E2 -21281.91} C_VEL
LIN {X 0,Y 242.361,Z 266.621,A -85,B 0,C 180,E1 -21284.104,E2 -21284.104} C_VEL
LIN {X 0,Y 242.844,Z 267.537,A -85,B 0,C 180,E1 -21286.345,E2 -21286.345} C_VEL
LIN {X 0,Y 243.326,Z 269.307,A -85,B 0,C 180,E1 -21288.674,E2 -21288.674} C_VEL
LIN {X 0,Y 243.775,Z 271.987,A -85,B 0,C 180,E1 -21291.115,E2 -21291.115} C_VEL
LIN {X 0,Y 243.831,Z 273.435,A -85,B 0,C 180,E1 -21292.114,E2 -21292.114} C_VEL
LIN {X 0,Y 243.613,Z 274.527,A -85,B 0,C 180,E1 -21292.709,E2 -21292.709} C_VEL
LIN {X 0,Y 240.366,Z 280.692,A -85,B 0,C 180,E1 -21294.954,E2 -21294.954} C_VEL
LIN {X 0,Y 238.071,Z 283.753,A -85,B 0,C 180,E1 -21295.88,E2 -21295.88} C_VEL
LIN {X 0,Y 232.065,Z 290.386,A -85,B 0,C 180,E1 -21297.992,E2 -21297.992} C_VEL
LIN {X 0,Y 226.551,Z 295.855,A -85,B 0,C 180,E1 -21300.239,E2 -21300.239} C_VEL
LIN {X 0,Y 221.418,Z 300.445,A -85,B 0,C 180,E1 -21302.717,E2 -21302.717} C_VEL
LIN {X 0,Y 217.197,Z 303.792,A -85,B 0,C 180,E1 -21305.121,E2 -21305.121} C_VEL
LIN {X 0,Y 212.623,Z 307.128,A -85,B 0,C 180,E1 -21308.676,E2 -21308.676} C_VEL
LIN {X 0,Y 210.967,Z 308.051,A -85,B 0,C 180,E1 -21310.177,E2 -21310.177} C_VEL
LIN {X 0,Y 208.844,Z 308.8,A -85,B 0,C 180,E1 -21311.669,E2 -21311.669} C_VEL
LIN {X 0,Y 204.087,Z 309.24,A -85,B 0,C 180,E1 -21314.08,E2 -21314.08} C_VEL
LIN {X 0,Y 199.872,Z 308.836,A -85,B 0,C 180,E1 -21316.615,E2 -21316.615} C_VEL
LIN {X 0,Y 198.636,Z 308.28,A -85,B 0,C 180,E1 -21318.263,E2 -21318.263} C_VEL
LIN {X 0,Y 198.07,Z 306.6,A -85,B 0,C 180,E1 -21321.837,E2 -21321.837} C_VEL
LIN {X 0,Y 198.148,Z 305.153,A -85,B 0,C 180,E1 -21323.889,E2 -21323.889} C_VEL
LIN {X 0,Y 198.846,Z 300.988,A -85,B 0,C 180,E1 -21327.971,E2 -21327.971} C_VEL
LIN {X 0,Y 199.182,Z 298.176,A -85,B 0,C 180,E1 -21329.997,E2 -21329.997} C_VEL
LIN {X 0,Y 199.251,Z 292.673,A -85,B 0,C 180,E1 -21333.03,E2 -21333.03} C_VEL
LIN {X 0,Y 199.333,Z 286.875,A -85,B 0,C 180,E1 -21335.561,E2 -21335.561} C_VEL
LIN {X 0,Y 199.364,Z 279.636,A -85,B 0,C 180,E1 -21338.103,E2 -21338.103} C_VEL
LIN {X 0,Y 199.717,Z 270.824,A -85,B 0,C 180,E1 -21340.643,E2 -21340.643} C_VEL
LIN {X 0,Y 200.208,Z 260.923,A -85,B 0,C 180,E1 -21342.928,E2 -21342.928} C_VEL
LIN {X 0,Y 200.848,Z 249.942,A -85,B 0,C 180,E1 -21344.952,E2 -21344.952} C_VEL
LIN {X 0,Y 200.872,Z 244.747,A -85,B 0,C 180,E1 -21345.729,E2 -21345.729} C_VEL
LIN {X 0,Y 199.658,Z 232.007,A -85,B 0,C 180,E1 -21347.252,E2 -21347.252} C_VEL
LIN {X 0,Y 199.185,Z 219.833,A -85,B 0,C 180,E1 -21348.35,E2 -21348.35} C_VEL
LIN {X 0,Y 201.097,Z 208.093,A -85,B 0,C 180,E1 -21355.899,E2 -21355.899} C_VEL
LIN {X 0,Y 202.426,Z 203.099,A -85,B 0,C 180,E1 -21359.078,E2 -21359.078} C_VEL
LIN {X 0,Y 202.45,Z 200.831,A -85,B 0,C 180,E1 -21360.54,E2 -21360.54} C_VEL
LIN {X 0,Y 200.986,Z 193.959,A -85,B 0,C 180,E1 -21365.129,E2 -21365.129} C_VEL
LIN {X 0,Y 199.773,Z 187.595,A -85,B 0,C 180,E1 -21369.667,E2 -21369.667} C_VEL
LIN {X 0,Y 199.638,Z 187.614,A -85,B 0,C 180,E1 -21375.245,E2 -21375.245} C_VEL
LIN {X 0,Y 199.657,Z 187.611,A -85,B 0,C 180,E1 -21378.025,E2 -21378.025} C_VEL
LIN {X 0,Y 199.671,Z 187.613,A -85,B 0,C 180,E1 -21380.74,E2 -21380.74} C_VEL
LIN {X 0,Y 199.624,Z 187.615,A -85,B 0,C 180,E1 -21385.715,E2 -21385.715} C_VEL
LIN {X 0,Y 199.686,Z 187.612,A -85,B 0,C 180,E1 -21388.134,E2 -21388.134} C_VEL
LIN {X 0,Y 199.674,Z 187.609,A -85,B 0,C 180,E1 -21392.77,E2 -21392.77} C_VEL
LIN {X 0,Y 199.703,Z 187.608,A -85,B 0,C 180,E1 -21397.225,E2 -21397.225} C_VEL
LIN {X 0,Y 199.784,Z 187.596,A -85,B 0,C 180,E1 -21401.757,E2 -21401.757} C_VEL
LIN {X 0,Y 199.836,Z 187.593,A -85,B 0,C 180,E1 -21405.748,E2 -21405.748} C_VEL
LIN {X 0,Y 200.058,Z 187.562,A -85,B 0,C 180,E1 -21409.883,E2 -21409.883} C_VEL
LIN {X 0,Y 200.023,Z 187.567,A -85,B 0,C 180,E1 -21413.949,E2 -21413.949} C_VEL
LIN {X 0,Y 200.312,Z 187.53,A -85,B 0,C 180,E1 -21417.989,E2 -21417.989} C_VEL
LIN {X 0,Y 200.466,Z 187.508,A -85,B 0,C 180,E1 -21420,E2 -21420} C_VEL
LIN {X 0,Y 200.015,Z 187.569,A -85,B 0,C 180,E1 -21424.03,E2 -21424.03} C_VEL
LIN {X 0,Y 200.099,Z 187.556,A -85,B 0,C 180,E1 -21428.076,E2 -21428.076} C_VEL
LIN {X 0,Y 199.901,Z 187.584,A -85,B 0,C 180,E1 -21432.178,E2 -21432.178} C_VEL
LIN {X 0,Y 199.792,Z 187.596,A -85,B 0,C 180,E1 -21436.344,E2 -21436.344} C_VEL
LIN {X 0,Y 199.679,Z 187.612,A -85,B 0,C 180,E1 -21440.607,E2 -21440.607} C_VEL
LIN {X 0,Y 199.639,Z 187.612,A -85,B 0,C 180,E1 -21444.989,E2 -21444.989} C_VEL
LIN {X 0,Y 199.597,Z 187.621,A -85,B 0,C 180,E1 -21449.535,E2 -21449.535} C_VEL
LIN {X 0,Y 199.64,Z 187.614,A -85,B 0,C 180,E1 -21452.348,E2 -21452.348} C_VEL
LIN {X 0,Y 199.63,Z 187.616,A -85,B 0,C 180,E1 -21456.762,E2 -21456.762} C_VEL
LIN {X 0,Y 199.631,Z 187.618,A -85,B 0,C 180,E1 -21459.323,E2 -21459.323} C_VEL
LIN {X 0,Y 199.591,Z 187.618,A -85,B 0,C 180,E1 -21462.321,E2 -21462.321} C_VEL
LIN {X 0,Y 199.586,Z 187.622,A -85,B 0,C 180,E1 -21465.236,E2 -21465.236} C_VEL
LIN {X 0,Y 199.572,Z 187.624,A -85,B 0,C 180,E1 -21468.008,E2 -21468.008} C_VEL
LIN {X 0,Y 199.603,Z 187.618,A -85,B 0,C 180,E1 -21470.77,E2 -21470.77} C_VEL
LIN {X 0,Y 199.607,Z 187.62,A -85,B 0,C 180,E1 -21475.717,E2 -21475.717} C_VEL
LIN {X 0,Y 199.695,Z 187.607,A -85,B 0,C 180,E1 -21478.14,E2 -21478.14} C_VEL
LIN {X 0,Y 199.683,Z 187.611,A -85,B 0,C 180,E1 -21482.775,E2 -21482.775} C_VEL
LIN {X 0,Y 199.735,Z 187.602,A -85,B 0,C 180,E1 -21487.232,E2 -21487.232} C_VEL
LIN {X 0,Y 199.835,Z 187.591,A -85,B 0,C 180,E1 -21491.725,E2 -21491.725} C_VEL
LIN {X 0,Y 199.835,Z 187.59,A -85,B 0,C 180,E1 -21495.752,E2 -21495.752} C_VEL
LIN {X 0,Y 200.075,Z 187.561,A -85,B 0,C 180,E1 -21499.888,E2 -21499.888} C_VEL
LIN {X 0,Y 200.132,Z 187.556,A -85,B 0,C 180,E1 -21501.928,E2 -21501.928} C_VEL
LIN {X 0,Y 200.322,Z 187.531,A -85,B 0,C 180,E1 -21507.993,E2 -21507.993} C_VEL
LIN {X 0,Y 200.452,Z 187.518,A -85,B 0,C 180,E1 -21510.003,E2 -21510.003} C_VEL
LIN {X 0,Y 200.321,Z 187.532,A -85,B 0,C 180,E1 -21512.014,E2 -21512.014} C_VEL
LIN {X 0,Y 200.135,Z 187.555,A -85,B 0,C 180,E1 -21518.078,E2 -21518.078} C_VEL
LIN {X 0,Y 199.91,Z 187.578,A -85,B 0,C 180,E1 -21522.18,E2 -21522.18} C_VEL
LIN {X 0,Y 199.809,Z 187.594,A -85,B 0,C 180,E1 -21526.346,E2 -21526.346} C_VEL
LIN {X 0,Y 199.68,Z 187.608,A -85,B 0,C 180,E1 -21530.611,E2 -21530.611} C_VEL
LIN {X 0,Y 199.63,Z 187.619,A -85,B 0,C 180,E1 -21534.993,E2 -21534.993} C_VEL
LIN {X 0,Y 199.612,Z 187.615,A -85,B 0,C 180,E1 -21539.536,E2 -21539.536} C_VEL
LIN {X 0,Y 199.671,Z 187.611,A -85,B 0,C 180,E1 -21542.355,E2 -21542.355} C_VEL
LIN {X 0,Y 199.626,Z 187.618,A -85,B 0,C 180,E1 -21546.766,E2 -21546.766} C_VEL
LIN {X 0,Y 199.602,Z 187.618,A -85,B 0,C 180,E1 -21549.333,E2 -21549.333} C_VEL
LIN {X 0,Y 199.573,Z 187.625,A -85,B 0,C 180,E1 -21552.31,E2 -21552.31} C_VEL
LIN {X 0,Y 199.584,Z 187.621,A -85,B 0,C 180,E1 -21555.23,E2 -21555.23} C_VEL
LIN {X 0,Y 199.682,Z 187.611,A -85,B 0,C 180,E1 -21560.747,E2 -21560.747} C_VEL
LIN {X 0,Y 199.989,Z 187.69,A -85,B 0,C 180,E1 -21564.869,E2 -21564.869} C_VEL
LIN {X 0,Y 200.592,Z 190.541,A -85,B 0,C 180,E1 -21567.237,E2 -21567.237} C_VEL
LIN {X 0,Y 200.557,Z 193.314,A -85,B 0,C 180,E1 -21569.462,E2 -21569.462} C_VEL
LIN {X 0,Y 199.598,Z 198.947,A -85,B 0,C 180,E1 -21573.888,E2 -21573.888} C_VEL
LIN {X 0,Y 198.861,Z 204.494,A -85,B 0,C 180,E1 -21578.218,E2 -21578.218} C_VEL
LIN {X 0,Y 198.145,Z 211.299,A -85,B 0,C 180,E1 -21583.516,E2 -21583.516} C_VEL
LIN {X 0,Y 198.063,Z 217.492,A -85,B 0,C 180,E1 -21588.292,E2 -21588.292} C_VEL
LIN {X 0,Y 198.624,Z 228.33,A -85,B 0,C 180,E1 -21589.552,E2 -21589.552} C_VEL
LIN {X 0,Y 199.374,Z 236.807,A -85,B 0,C 180,E1 -21590.771,E2 -21590.771} C_VEL
LIN {X 0,Y 198.945,Z 247.55,A -85,B 0,C 180,E1 -21592.743,E2 -21592.743} C_VEL
LIN {X 0,Y 198.502,Z 256.996,A -85,B 0,C 180,E1 -21594.922,E2 -21594.922} C_VEL
LIN {X 0,Y 198.303,Z 264.264,A -85,B 0,C 180,E1 -21596.953,E2 -21596.953} C_VEL
LIN {X 0,Y 197.965,Z 271.659,A -85,B 0,C 180,E1 -21599.492,E2 -21599.492} C_VEL
LIN {X 0,Y 198.024,Z 278.78,A -85,B 0,C 180,E1 -21602.543,E2 -21602.543} C_VEL
LIN {X 0,Y 198.543,Z 283.492,A -85,B 0,C 180,E1 -21605.077,E2 -21605.077} C_VEL
LIN {X 0,Y 199.79,Z 287.878,A -85,B 0,C 180,E1 -21608.089,E2 -21608.089} C_VEL
LIN {X 0,Y 200.687,Z 290.111,A -85,B 0,C 180,E1 -21610.085,E2 -21610.085} C_VEL
LIN {X 0,Y 202.033,Z 291.8,A -85,B 0,C 180,E1 -21612.047,E2 -21612.047} C_VEL
LIN {X 0,Y 203.673,Z 293.019,A -85,B 0,C 180,E1 -21613.978,E2 -21613.978} C_VEL
LIN {X 0,Y 205.743,Z 293.73,A -85,B 0,C 180,E1 -21615.859,E2 -21615.859} C_VEL
LIN {X 0,Y 207.986,Z 293.955,A -85,B 0,C 180,E1 -21617.705,E2 -21617.705} C_VEL
LIN {X 0,Y 210.577,Z 293.701,A -85,B 0,C 180,E1 -21619.497,E2 -21619.497} C_VEL
LIN {X 0,Y 213.502,Z 292.939,A -85,B 0,C 180,E1 -21621.229,E2 -21621.229} C_VEL
LIN {X 0,Y 216.704,Z 291.714,A -85,B 0,C 180,E1 -21622.903,E2 -21622.903} C_VEL
LIN {X 0,Y 221.833,Z 288.939,A -85,B 0,C 180,E1 -21625.322,E2 -21625.322} C_VEL
LIN {X 0,Y 225.419,Z 286.526,A -85,B 0,C 180,E1 -21626.877,E2 -21626.877} C_VEL
LIN {X 0,Y 227.901,Z 284.125,A -85,B 0,C 180,E1 -21628.554,E2 -21628.554} C_VEL
LIN {X 0,Y 231.593,Z 279.538,A -85,B 0,C 180,E1 -21631.817,E2 -21631.817} C_VEL
LIN {X 0,Y 234.342,Z 275.567,A -85,B 0,C 180,E1 -21634.738,E2 -21634.738} C_VEL
LIN {X 0,Y 235.569,Z 273.545,A -85,B 0,C 180,E1 -21636.633,E2 -21636.633} C_VEL
LIN {X 0,Y 236.483,Z 271.848,A -85,B 0,C 180,E1 -21639.401,E2 -21639.401} C_VEL
LIN {X 0,Y 236.786,Z 271.451,A -85,B 0,C 180,E1 -21640.767,E2 -21640.767} C_VEL
LIN {X 0,Y 237.116,Z 271.445,A -85,B 0,C 180,E1 -21642.978,E2 -21642.978} C_VEL
LIN {X 0,Y 237.525,Z 272.048,A -85,B 0,C 180,E1 -21645.245,E2 -21645.245} C_VEL
LIN {X 0,Y 237.917,Z 273.381,A -85,B 0,C 180,E1 -21647.604,E2 -21647.604} C_VEL
LIN {X 0,Y 238.317,Z 275.53,A -85,B 0,C 180,E1 -21650.063,E2 -21650.063} C_VEL
LIN {X 0,Y 238.287,Z 277.59,A -85,B 0,C 180,E1 -21651.727,E2 -21651.727} C_VEL
LIN {X 0,Y 236.655,Z 280.597,A -85,B 0,C 180,E1 -21653.029,E2 -21653.029} C_VEL
LIN {X 0,Y 234.865,Z 283.265,A -85,B 0,C 180,E1 -21654.054,E2 -21654.054} C_VEL
LIN {X 0,Y 228.212,Z 290.214,A -85,B 0,C 180,E1 -21656.333,E2 -21656.333} C_VEL
LIN {X 0,Y 222.553,Z 295.401,A -85,B 0,C 180,E1 -21658.488,E2 -21658.488} C_VEL
LIN {X 0,Y 217.041,Z 299.914,A -85,B 0,C 180,E1 -21660.938,E2 -21660.938} C_VEL
LIN {X 0,Y 213.771,Z 302.312,A -85,B 0,C 180,E1 -21662.593,E2 -21662.593} C_VEL
LIN {X 0,Y 210.792,Z 304.284,A -85,B 0,C 180,E1 -21664.312,E2 -21664.312} C_VEL
LIN {X 0,Y 206.025,Z 307.19,A -85,B 0,C 180,E1 -21667.958,E2 -21667.958} C_VEL
LIN {X 0,Y 202.163,Z 308.7,A -85,B 0,C 180,E1 -21671.764,E2 -21671.764} C_VEL
LIN {X 0,Y 199.568,Z 308.882,A -85,B 0,C 180,E1 -21675.726,E2 -21675.726} C_VEL
LIN {X 0,Y 198.636,Z 308.28,A -85,B 0,C 180,E1 -21678.263,E2 -21678.263} C_VEL
LIN {X 0,Y 197.604,Z 307.537,A -85,B 0,C 180,E1 -21679.929,E2 -21679.929} C_VEL
LIN {X 0,Y 194.562,Z 305.306,A -85,B 0,C 180,E1 -21682.612,E2 -21682.612} C_VEL
LIN {X 0,Y 192.342,Z 302.912,A -85,B 0,C 180,E1 -21684.776,E2 -21684.776} C_VEL
LIN {X 0,Y 191.646,Z 300.911,A -85,B 0,C 180,E1 -21686.439,E2 -21686.439} C_VEL
LIN {X 0,Y 191.713,Z 300.239,A -85,B 0,C 180,E1 -21686.998,E2 -21686.998} C_VEL
LIN {X 0,Y 192.205,Z 297.736,A -85,B 0,C 180,E1 -21688.949,E2 -21688.949} C_VEL
LIN {X 0,Y 192.378,Z 294.348,A -85,B 0,C 180,E1 -21691.043,E2 -21691.043} C_VEL
LIN {X 0,Y 192.462,Z 287.976,A -85,B 0,C 180,E1 -21694.185,E2 -21694.185} C_VEL
LIN {X 0,Y 192.502,Z 281.232,A -85,B 0,C 180,E1 -21696.811,E2 -21696.811} C_VEL
LIN {X 0,Y 192.717,Z 271.948,A -85,B 0,C 180,E1 -21699.709,E2 -21699.709} C_VEL
LIN {X 0,Y 193.157,Z 262.584,A -85,B 0,C 180,E1 -21702.073,E2 -21702.073} C_VEL
LIN {X 0,Y 193.775,Z 250.63,A -85,B 0,C 180,E1 -21704.435,E2 -21704.435} C_VEL
LIN {X 0,Y 193.893,Z 244.805,A -85,B 0,C 180,E1 -21705.367,E2 -21705.367} C_VEL
LIN {X 0,Y 192.632,Z 231.999,A -85,B 0,C 180,E1 -21706.966,E2 -21706.966} C_VEL
LIN {X 0,Y 192.142,Z 219.834,A -85,B 0,C 180,E1 -21708.1,E2 -21708.1} C_VEL
LIN {X 0,Y 194.329,Z 206.787,A -85,B 0,C 180,E1 -21716.872,E2 -21716.872} C_VEL
LIN {X 0,Y 195.273,Z 203.484,A -85,B 0,C 180,E1 -21719.066,E2 -21719.066} C_VEL
LIN {X 0,Y 195.421,Z 201.588,A -85,B 0,C 180,E1 -21720.33,E2 -21720.33} C_VEL
LIN {X 0,Y 193.84,Z 194.2,A -85,B 0,C 180,E1 -21725.454,E2 -21725.454} C_VEL
LIN {X 0,Y 192.742,Z 188.471,A -85,B 0,C 180,E1 -21729.585,E2 -21729.585} C_VEL
LIN {X 0,Y 192.585,Z 188.494,A -85,B 0,C 180,E1 -21736.103,E2 -21736.103} C_VEL
LIN {X 0,Y 192.582,Z 188.495,A -85,B 0,C 180,E1 -21740.023,E2 -21740.023} C_VEL
LIN {X 0,Y 192.592,Z 188.493,A -85,B 0,C 180,E1 -21744.277,E2 -21744.277} C_VEL
LIN {X 0,Y 192.589,Z 188.494,A -85,B 0,C 180,E1 -21749.277,E2 -21749.277} C_VEL
LIN {X 0,Y 192.65,Z 188.488,A -85,B 0,C 180,E1 -21751.689,E2 -21751.689} C_VEL
LIN {X 0,Y 192.674,Z 188.483,A -85,B 0,C 180,E1 -21756.344,E2 -21756.344} C_VEL
LIN {X 0,Y 192.72,Z 188.478,A -85,B 0,C 180,E1 -21761.457,E2 -21761.457} C_VEL
LIN {X 0,Y 192.76,Z 188.473,A -85,B 0,C 180,E1 -21765.213,E2 -21765.213} C_VEL
LIN {X 0,Y 192.969,Z 188.446,A -85,B 0,C 180,E1 -21769.508,E2 -21769.508} C_VEL
LIN {X 0,Y 193.049,Z 188.435,A -85,B 0,C 180,E1 -21771.627,E2 -21771.627} C_VEL
LIN {X 0,Y 193.254,Z 188.41,A -85,B 0,C 180,E1 -21777.916,E2 -21777.916} C_VEL
LIN {X 0,Y 193.43,Z 188.384,A -85,B 0,C 180,E1 -21780,E2 -21780} C_VEL
LIN {X 0,Y 192.962,Z 188.448,A -85,B 0,C 180,E1 -21784.177,E2 -21784.177} C_VEL
LIN {X 0,Y 193.049,Z 188.435,A -85,B 0,C 180,E1 -21788.373,E2 -21788.373} C_VEL
LIN {X 0,Y 192.841,Z 188.465,A -85,B 0,C 180,E1 -21792.631,E2 -21792.631} C_VEL
LIN {X 0,Y 192.746,Z 188.471,A -85,B 0,C 180,E1 -21796.96,E2 -21796.96} C_VEL
LIN {X 0,Y 192.609,Z 188.491,A -85,B 0,C 180,E1 -21801.4,E2 -21801.4} C_VEL
LIN {X 0,Y 192.628,Z 188.489,A -85,B 0,C 180,E1 -21804.21,E2 -21804.21} C_VEL
LIN {X 0,Y 192.591,Z 188.494,A -85,B 0,C 180,E1 -21808.868,E2 -21808.868} C_VEL
LIN {X 0,Y 192.585,Z 188.492,A -85,B 0,C 180,E1 -21813.188,E2 -21813.188} C_VEL
LIN {X 0,Y 192.6,Z 188.492,A -85,B 0,C 180,E1 -21816.61,E2 -21816.61} C_VEL
LIN {X 0,Y 192.527,Z 188.501,A -85,B 0,C 180,E1 -21821.077,E2 -21821.077} C_VEL
LIN {X 0,Y 192.513,Z 188.504,A -85,B 0,C 180,E1 -21826.087,E2 -21826.087} C_VEL
LIN {X 0,Y 192.511,Z 188.501,A -85,B 0,C 180,E1 -21830.054,E2 -21830.054} C_VEL
LIN {X 0,Y 192.554,Z 188.498,A -85,B 0,C 180,E1 -21834.273,E2 -21834.273} C_VEL
LIN {X 0,Y 192.604,Z 188.494,A -85,B 0,C 180,E1 -21837.061,E2 -21837.061} C_VEL
LIN {X 0,Y 192.66,Z 188.484,A -85,B 0,C 180,E1 -21841.695,E2 -21841.695} C_VEL
LIN {X 0,Y 192.702,Z 188.48,A -85,B 0,C 180,E1 -21846.352,E2 -21846.352} C_VEL
LIN {X 0,Y 192.779,Z 188.47,A -85,B 0,C 180,E1 -21851.417,E2 -21851.417} C_VEL
LIN {X 0,Y 192.821,Z 188.461,A -85,B 0,C 180,E1 -21857.371,E2 -21857.371} C_VEL
LIN {X 0,Y 193.019,Z 188.439,A -85,B 0,C 180,E1 -21859.514,E2 -21859.514} C_VEL
LIN {X 0,Y 193.005,Z 188.442,A -85,B 0,C 180,E1 -21863.732,E2 -21863.732} C_VEL
LIN {X 0,Y 193.264,Z 188.41,A -85,B 0,C 180,E1 -21867.919,E2 -21867.919} C_VEL
LIN {X 0,Y 193.42,Z 188.394,A -85,B 0,C 180,E1 -21870.003,E2 -21870.003} C_VEL
LIN {X 0,Y 192.977,Z 188.443,A -85,B 0,C 180,E1 -21874.18,E2 -21874.18} C_VEL
LIN {X 0,Y 193.082,Z 188.433,A -85,B 0,C 180,E1 -21878.375,E2 -21878.375} C_VEL
LIN {X 0,Y 193.013,Z 188.44,A -85,B 0,C 180,E1 -21880.541,E2 -21880.541} C_VEL
LIN {X 0,Y 192.761,Z 188.473,A -85,B 0,C 180,E1 -21886.962,E2 -21886.962} C_VEL
LIN {X 0,Y 192.602,Z 188.49,A -85,B 0,C 180,E1 -21891.405,E2 -21891.405} C_VEL
LIN {X 0,Y 192.624,Z 188.489,A -85,B 0,C 180,E1 -21894.197,E2 -21894.197} C_VEL
LIN {X 0,Y 192.605,Z 188.492,A -85,B 0,C 180,E1 -21898.868,E2 -21898.868} C_VEL
LIN {X 0,Y 192.6,Z 188.494,A -85,B 0,C 180,E1 -21903.189,E2 -21903.189} C_VEL
LIN {X 0,Y 192.549,Z 188.497,A -85,B 0,C 180,E1 -21908.356,E2 -21908.356} C_VEL
LIN {X 0,Y 192.492,Z 188.507,A -85,B 0,C 180,E1 -21913.096,E2 -21913.096} C_VEL
LIN {X 0,Y 192.498,Z 188.502,A -85,B 0,C 180,E1 -21916.906,E2 -21916.906} C_VEL
LIN {X 0,Y 192.645,Z 188.487,A -85,B 0,C 180,E1 -21921.67,E2 -21921.67} C_VEL
LIN {X 0,Y 192.952,Z 188.565,A -85,B 0,C 180,E1 -21924.971,E2 -21924.971} C_VEL
LIN {X 0,Y 193.592,Z 192.405,A -85,B 0,C 180,E1 -21928.238,E2 -21928.238} C_VEL
LIN {X 0,Y 192.935,Z 196.68,A -85,B 0,C 180,E1 -21931.735,E2 -21931.735} C_VEL
LIN {X 0,Y 191.897,Z 203.665,A -85,B 0,C 180,E1 -21937.384,E2 -21937.384} C_VEL
LIN {X 0,Y 191.09,Z 210.627,A -85,B 0,C 180,E1 -21942.997,E2 -21942.997} C_VEL
LIN {X 0,Y 191.025,Z 217.522,A -85,B 0,C 180,E1 -21948.527,E2 -21948.527} C_VEL
LIN {X 0,Y 191.702,Z 229.323,A -85,B 0,C 180,E1 -21949.98,E2 -21949.98} C_VEL
LIN {X 0,Y 192.355,Z 237.496,A -85,B 0,C 180,E1 -21951.225,E2 -21951.225} C_VEL
LIN {X 0,Y 191.845,Z 248.795,A -85,B 0,C 180,E1 -21953.434,E2 -21953.434} C_VEL
LIN {X 0,Y 191.485,Z 258.381,A -85,B 0,C 180,E1 -21955.791,E2 -21955.791} C_VEL
LIN {X 0,Y 191.198,Z 265.378,A -85,B 0,C 180,E1 -21957.894,E2 -21957.894} C_VEL
LIN {X 0,Y 190.989,Z 272.595,A -85,B 0,C 180,E1 -21960.527,E2 -21960.527} C_VEL
LIN {X 0,Y 191.191,Z 279.55,A -85,B 0,C 180,E1 -21963.688,E2 -21963.688} C_VEL
LIN {X 0,Y 191.873,Z 284.176,A -85,B 0,C 180,E1 -21966.309,E2 -21966.309} C_VEL
LIN {X 0,Y 193.24,Z 288.477,A -85,B 0,C 180,E1 -21969.42,E2 -21969.42} C_VEL
LIN {X 0,Y 195.112,Z 291.59,A -85,B 0,C 180,E1 -21972.482,E2 -21972.482} C_VEL
LIN {X 0,Y 196.806,Z 293.034,A -85,B 0,C 180,E1 -21974.476,E2 -21974.476} C_VEL
LIN {X 0,Y 198.944,Z 294.014,A -85,B 0,C 180,E1 -21976.416,E2 -21976.416} C_VEL
LIN {X 0,Y 201.251,Z 294.485,A -85,B 0,C 180,E1 -21978.318,E2 -21978.318} C_VEL
LIN {X 0,Y 203.94,Z 294.507,A -85,B 0,C 180,E1 -21980.158,E2 -21980.158} C_VEL
LIN {X 0,Y 206.95,Z 294.015,A -85,B 0,C 180,E1 -21981.935,E2 -21981.935} C_VEL
LIN {X 0,Y 210.261,Z 293.071,A -85,B 0,C 180,E1 -21983.647,E2 -21983.647} C_VEL
LIN {X 0,Y 213.758,Z 291.643,A -85,B 0,C 180,E1 -21985.304,E2 -21985.304} C_VEL
LIN {X 0,Y 219.342,Z 288.652,A -85,B 0,C 180,E1 -21987.684,E2 -21987.684} C_VEL
LIN {X 0,Y 220.857,Z 287.551,A -85,B 0,C 180,E1 -21988.511,E2 -21988.511} C_VEL
LIN {X 0,Y 224.289,Z 284.383,A -85,B 0,C 180,E1 -21991.133,E2 -21991.133} C_VEL
LIN {X 0,Y 227.28,Z 281.111,A -85,B 0,C 180,E1 -21993.821,E2 -21993.821} C_VEL
LIN {X 0,Y 229.067,Z 279.027,A -85,B 0,C 180,E1 -21995.658,E2 -21995.658} C_VEL
LIN {X 0,Y 230.306,Z 277.43,A -85,B 0,C 180,E1 -21997.613,E2 -21997.613} C_VEL
LIN {X 0,Y 231.143,Z 276.403,A -85,B 0,C 180,E1 -21999.681,E2 -21999.681} C_VEL
LIN {X 0,Y 231.596,Z 276.085,A -85,B 0,C 180,E1 -22001.883,E2 -22001.883} C_VEL
LIN {X 0,Y 231.986,Z 276.394,A -85,B 0,C 180,E1 -22004.17,E2 -22004.17} C_VEL
LIN {X 0,Y 232.358,Z 277.367,A -85,B 0,C 180,E1 -22006.545,E2 -22006.545} C_VEL
LIN {X 0,Y 232.672,Z 279.104,A -85,B 0,C 180,E1 -22009.038,E2 -22009.038} C_VEL
LIN {X 0,Y 232.681,Z 280.652,A -85,B 0,C 180,E1 -22010.63,E2 -22010.63} C_VEL
LIN {X 0,Y 232.043,Z 282.223,A -85,B 0,C 180,E1 -22011.617,E2 -22011.617} C_VEL
LIN {X 0,Y 229.219,Z 285.835,A -85,B 0,C 180,E1 -22013.14,E2 -22013.14} C_VEL
LIN {X 0,Y 222.469,Z 292.007,A -85,B 0,C 180,E1 -22015.342,E2 -22015.342} C_VEL
LIN {X 0,Y 216.147,Z 297.095,A -85,B 0,C 180,E1 -22017.714,E2 -22017.714} C_VEL
LIN {X 0,Y 210.926,Z 300.798,A -85,B 0,C 180,E1 -22020.01,E2 -22020.01} C_VEL
LIN {X 0,Y 207.54,Z 302.942,A -85,B 0,C 180,E1 -22021.697,E2 -22021.697} C_VEL
LIN {X 0,Y 204.442,Z 304.686,A -85,B 0,C 180,E1 -22023.452,E2 -22023.452} C_VEL
LIN {X 0,Y 199.464,Z 307.132,A -85,B 0,C 180,E1 -22027.193,E2 -22027.193} C_VEL
LIN {X 0,Y 195.437,Z 308.266,A -85,B 0,C 180,E1 -22031.113,E2 -22031.113} C_VEL
LIN {X 0,Y 192.723,Z 308.047,A -85,B 0,C 180,E1 -22035.207,E2 -22035.207} C_VEL
LIN {X 0,Y 191.374,Z 306.559,A -85,B 0,C 180,E1 -22039.416,E2 -22039.416} C_VEL
LIN {X 0,Y 191.229,Z 303.643,A -85,B 0,C 180,E1 -22043.667,E2 -22043.667} C_VEL
LIN {X 0,Y 191.713,Z 300.239,A -85,B 0,C 180,E1 -22046.998,E2 -22046.998} C_VEL
LIN {X 0,Y 191.676,Z 298.814,A -85,B 0,C 180,E1 -22048.086,E2 -22048.086} C_VEL
LIN {X 0,Y 190.65,Z 296.195,A -85,B 0,C 180,E1 -22049.644,E2 -22049.644} C_VEL
LIN {X 0,Y 188.998,Z 293.132,A -85,B 0,C 180,E1 -22051.116,E2 -22051.116} C_VEL
LIN {X 0,Y 186.712,Z 288.559,A -85,B 0,C 180,E1 -22053.053,E2 -22053.053} C_VEL
LIN {X 0,Y 185.72,Z 284.879,A -85,B 0,C 180,E1 -22054.511,E2 -22054.511} C_VEL
LIN {X 0,Y 185.646,Z 283.623,A -85,B 0,C 180,E1 -22055.002,E2 -22055.002} C_VEL
LIN {X 0,Y 185.632,Z 276.377,A -85,B 0,C 180,E1 -22057.611,E2 -22057.611} C_VEL
LIN {X 0,Y 185.949,Z 267.086,A -85,B 0,C 180,E1 -22060.346,E2 -22060.346} C_VEL
LIN {X 0,Y 186.431,Z 256.628,A -85,B 0,C 180,E1 -22062.792,E2 -22062.792} C_VEL
LIN {X 0,Y 187.017,Z 246.502,A -85,B 0,C 180,E1 -22064.691,E2 -22064.691} C_VEL
LIN {X 0,Y 185.864,Z 234.541,A -85,B 0,C 180,E1 -22066.33,E2 -22066.33} C_VEL
LIN {X 0,Y 185.135,Z 222.266,A -85,B 0,C 180,E1 -22067.604,E2 -22067.604} C_VEL
LIN {X 0,Y 185.091,Z 219.785,A -85,B 0,C 180,E1 -22067.848,E2 -22067.848} C_VEL
LIN {X 0,Y 187.151,Z 207.094,A -85,B 0,C 180,E1 -22076.78,E2 -22076.78} C_VEL
LIN {X 0,Y 188.283,Z 202.588,A -85,B 0,C 180,E1 -22079.893,E2 -22079.893} C_VEL
LIN {X 0,Y 187.519,Z 198.339,A -85,B 0,C 180,E1 -22082.914,E2 -22082.914} C_VEL
LIN {X 0,Y 185.921,Z 190.492,A -85,B 0,C 180,E1 -22088.703,E2 -22088.703} C_VEL
LIN {X 0,Y 185.709,Z 189.347,A -85,B 0,C 180,E1 -22089.714,E2 -22089.714} C_VEL
LIN {X 0,Y 185.546,Z 189.37,A -85,B 0,C 180,E1 -22096.021,E2 -22096.021} C_VEL
LIN {X 0,Y 185.533,Z 189.373,A -85,B 0,C 180,E1 -22099.912,E2 -22099.912} C_VEL
LIN {X 0,Y 185.551,Z 189.371,A -85,B 0,C 180,E1 -22102.697,E2 -22102.697} C_VEL
LIN {X 0,Y 185.531,Z 189.373,A -85,B 0,C 180,E1 -22107.972,E2 -22107.972} C_VEL
LIN {X 0,Y 185.57,Z 189.369,A -85,B 0,C 180,E1 -22110.575,E2 -22110.575} C_VEL
LIN {X 0,Y 185.569,Z 189.365,A -85,B 0,C 180,E1 -22115.38,E2 -22115.38} C_VEL
LIN {X 0,Y 185.663,Z 189.356,A -85,B 0,C 180,E1 -22121.132,E2 -22121.132} C_VEL
LIN {X 0,Y 185.752,Z 189.346,A -85,B 0,C 180,E1 -22126.879,E2 -22126.879} C_VEL
LIN {X 0,Y 185.996,Z 189.313,A -85,B 0,C 180,E1 -22131.307,E2 -22131.307} C_VEL
LIN {X 0,Y 186.198,Z 189.289,A -85,B 0,C 180,E1 -22137.837,E2 -22137.837} C_VEL
LIN {X 0,Y 186.394,Z 189.26,A -85,B 0,C 180,E1 -22140,E2 -22140} C_VEL
LIN {X 0,Y 185.909,Z 189.327,A -85,B 0,C 180,E1 -22144.336,E2 -22144.336} C_VEL
LIN {X 0,Y 185.996,Z 189.313,A -85,B 0,C 180,E1 -22148.693,E2 -22148.693} C_VEL
LIN {X 0,Y 185.752,Z 189.346,A -85,B 0,C 180,E1 -22153.121,E2 -22153.121} C_VEL
LIN {X 0,Y 185.662,Z 189.356,A -85,B 0,C 180,E1 -22158.868,E2 -22158.868} C_VEL
LIN {X 0,Y 185.566,Z 189.366,A -85,B 0,C 180,E1 -22164.648,E2 -22164.648} C_VEL
LIN {X 0,Y 185.533,Z 189.373,A -85,B 0,C 180,E1 -22169.501,E2 -22169.501} C_VEL
LIN {X 0,Y 185.507,Z 189.372,A -85,B 0,C 180,E1 -22174.63,E2 -22174.63} C_VEL
LIN {X 0,Y 185.534,Z 189.373,A -85,B 0,C 180,E1 -22177.306,E2 -22177.306} C_VEL
LIN {X 0,Y 185.486,Z 189.378,A -85,B 0,C 180,E1 -22180.736,E2 -22180.736} C_VEL
LIN {X 0,Y 185.479,Z 189.38,A -85,B 0,C 180,E1 -22186.049,E2 -22186.049} C_VEL
LIN {X 0,Y 185.461,Z 189.38,A -85,B 0,C 180,E1 -22189.898,E2 -22189.898} C_VEL
LIN {X 0,Y 185.499,Z 189.374,A -85,B 0,C 180,E1 -22192.714,E2 -22192.714} C_VEL
LIN {X 0,Y 185.54,Z 189.37,A -85,B 0,C 180,E1 -22197.979,E2 -22197.979} C_VEL
LIN {X 0,Y 185.577,Z 189.363,A -85,B 0,C 180,E1 -22200.579,E2 -22200.579} C_VEL
LIN {X 0,Y 185.584,Z 189.367,A -85,B 0,C 180,E1 -22205.386,E2 -22205.386} C_VEL
LIN {X 0,Y 185.691,Z 189.354,A -85,B 0,C 180,E1 -22211.119,E2 -22211.119} C_VEL
LIN {X 0,Y 185.741,Z 189.343,A -85,B 0,C 180,E1 -22216.882,E2 -22216.882} C_VEL
LIN {X 0,Y 186.029,Z 189.311,A -85,B 0,C 180,E1 -22221.312,E2 -22221.312} C_VEL
LIN {X 0,Y 186.209,Z 189.288,A -85,B 0,C 180,E1 -22227.84,E2 -22227.84} C_VEL
LIN {X 0,Y 186.386,Z 189.27,A -85,B 0,C 180,E1 -22230.003,E2 -22230.003} C_VEL
LIN {X 0,Y 185.925,Z 189.321,A -85,B 0,C 180,E1 -22234.339,E2 -22234.339} C_VEL
LIN {X 0,Y 186.032,Z 189.311,A -85,B 0,C 180,E1 -22238.695,E2 -22238.695} C_VEL
LIN {X 0,Y 185.746,Z 189.343,A -85,B 0,C 180,E1 -22243.125,E2 -22243.125} C_VEL
LIN {X 0,Y 185.693,Z 189.354,A -85,B 0,C 180,E1 -22247.628,E2 -22247.628} C_VEL
LIN {X 0,Y 185.562,Z 189.366,A -85,B 0,C 180,E1 -22252.259,E2 -22252.259} C_VEL
LIN {X 0,Y 185.504,Z 189.379,A -85,B 0,C 180,E1 -22257.045,E2 -22257.045} C_VEL
LIN {X 0,Y 185.548,Z 189.367,A -85,B 0,C 180,E1 -22259.502,E2 -22259.502} C_VEL
LIN {X 0,Y 185.503,Z 189.379,A -85,B 0,C 180,E1 -22264.635,E2 -22264.635} C_VEL
LIN {X 0,Y 185.506,Z 189.373,A -85,B 0,C 180,E1 -22267.317,E2 -22267.317} C_VEL
LIN {X 0,Y 185.468,Z 189.382,A -85,B 0,C 180,E1 -22270.724,E2 -22270.724} C_VEL
LIN {X 0,Y 185.466,Z 189.38,A -85,B 0,C 180,E1 -22276.057,E2 -22276.057} C_VEL
LIN {X 0,Y 185.518,Z 189.375,A -85,B 0,C 180,E1 -22279.908,E2 -22279.908} C_VEL
LIN {X 0,Y 185.939,Z 189.451,A -85,B 0,C 180,E1 -22285.132,E2 -22285.132} C_VEL
LIN {X 0,Y 186.532,Z 192.912,A -85,B 0,C 180,E1 -22288.165,E2 -22288.165} C_VEL
LIN {X 0,Y 185.843,Z 197.194,A -85,B 0,C 180,E1 -22291.79,E2 -22291.79} C_VEL
LIN {X 0,Y 184.754,Z 204.174,A -85,B 0,C 180,E1 -22297.642,E2 -22297.642} C_VEL
LIN {X 0,Y 184.048,Z 210.211,A -85,B 0,C 180,E1 -22302.686,E2 -22302.686} C_VEL
LIN {X 0,Y 184.023,Z 217.624,A -85,B 0,C 180,E1 -22308.852,E2 -22308.852} C_VEL
LIN {X 0,Y 184.758,Z 229.87,A -85,B 0,C 180,E1 -22310.414,E2 -22310.414} C_VEL
LIN {X 0,Y 185.352,Z 237.109,A -85,B 0,C 180,E1 -22311.551,E2 -22311.551} C_VEL
LIN {X 0,Y 184.893,Z 247.923,A -85,B 0,C 180,E1 -22313.726,E2 -22313.726} C_VEL
LIN {X 0,Y 184.536,Z 257.686,A -85,B 0,C 180,E1 -22316.179,E2 -22316.179} C_VEL
LIN {X 0,Y 184.232,Z 264.765,A -85,B 0,C 180,E1 -22318.361,E2 -22318.361} C_VEL
LIN {X 0,Y 184.031,Z 273.417,A -85,B 0,C 180,E1 -22321.641,E2 -22321.641} C_VEL
LIN {X 0,Y 184.433,Z 280.235,A -85,B 0,C 180,E1 -22324.919,E2 -22324.919} C_VEL
LIN {X 0,Y 185.34,Z 284.795,A -85,B 0,C 180,E1 -22327.627,E2 -22327.627} C_VEL
LIN {X 0,Y 186.804,Z 289.025,A -85,B 0,C 180,E1 -22330.843,E2 -22330.843} C_VEL
LIN {X 0,Y 188.206,Z 291.231,A -85,B 0,C 180,E1 -22332.947,E2 -22332.947} C_VEL
LIN {X 0,Y 189.957,Z 292.907,A -85,B 0,C 180,E1 -22335.01,E2 -22335.01} C_VEL
LIN {X 0,Y 192.167,Z 294.138,A -85,B 0,C 180,E1 -22337.013,E2 -22337.013} C_VEL
LIN {X 0,Y 194.539,Z 294.876,A -85,B 0,C 180,E1 -22338.974,E2 -22338.974} C_VEL
LIN {X 0,Y 197.332,Z 295.159,A -85,B 0,C 180,E1 -22340.864,E2 -22340.864} C_VEL
LIN {X 0,Y 200.422,Z 294.952,A -85,B 0,C 180,E1 -22342.689,E2 -22342.689} C_VEL
LIN {X 0,Y 203.853,Z 294.288,A -85,B 0,C 180,E1 -22344.438,E2 -22344.438} C_VEL
LIN {X 0,Y 207.468,Z 293.162,A -85,B 0,C 180,E1 -22346.128,E2 -22346.128} C_VEL
LIN {X 0,Y 211.319,Z 291.568,A -85,B 0,C 180,E1 -22347.75,E2 -22347.75} C_VEL
LIN {X 0,Y 214.918,Z 289.671,A -85,B 0,C 180,E1 -22349.375,E2 -22349.375} C_VEL
LIN {X 0,Y 217.417,Z 287.88,A -85,B 0,C 180,E1 -22351.145,E2 -22351.145} C_VEL
LIN {X 0,Y 221.44,Z 284.484,A -85,B 0,C 180,E1 -22354.389,E2 -22354.389} C_VEL
LIN {X 0,Y 223.684,Z 282.377,A -85,B 0,C 180,E1 -22356.653,E2 -22356.653} C_VEL
LIN {X 0,Y 224.921,Z 281.172,A -85,B 0,C 180,E1 -22358.677,E2 -22358.677} C_VEL
LIN {X 0,Y 225.772,Z 280.495,A -85,B 0,C 180,E1 -22360.822,E2 -22360.822} C_VEL
LIN {X 0,Y 226.214,Z 280.559,A -85,B 0,C 180,E1 -22363.118,E2 -22363.118} C_VEL
LIN {X 0,Y 226.572,Z 281.245,A -85,B 0,C 180,E1 -22365.515,E2 -22365.515} C_VEL
LIN {X 0,Y 226.802,Z 282.629,A -85,B 0,C 180,E1 -22368.048,E2 -22368.048} C_VEL
LIN {X 0,Y 226.857,Z 283.661,A -85,B 0,C 180,E1 -22369.412,E2 -22369.412} C_VEL
LIN {X 0,Y 226.112,Z 285.561,A -85,B 0,C 180,E1 -22370.992,E2 -22370.992} C_VEL
LIN {X 0,Y 223.525,Z 288.268,A -85,B 0,C 180,E1 -22372.182,E2 -22372.182} C_VEL
LIN {X 0,Y 216.79,Z 293.67,A -85,B 0,C 180,E1 -22374.298,E2 -22374.298} C_VEL
LIN {X 0,Y 208.572,Z 299.359,A -85,B 0,C 180,E1 -22377.372,E2 -22377.372} C_VEL
LIN {X 0,Y 200.611,Z 303.837,A -85,B 0,C 180,E1 -22381.143,E2 -22381.143} C_VEL
LIN {X 0,Y 195.369,Z 306.134,A -85,B 0,C 180,E1 -22384.423,E2 -22384.423} C_VEL
LIN {X 0,Y 190.65,Z 307.489,A -85,B 0,C 180,E1 -22388.365,E2 -22388.365} C_VEL
LIN {X 0,Y 187.07,Z 307.554,A -85,B 0,C 180,E1 -22392.506,E2 -22392.506} C_VEL
LIN {X 0,Y 185.033,Z 306.33,A -85,B 0,C 180,E1 -22396.824,E2 -22396.824} C_VEL
LIN {X 0,Y 184.266,Z 303.82,A -85,B 0,C 180,E1 -22401.221,E2 -22401.221} C_VEL
LIN {X 0,Y 184.463,Z 300.964,A -85,B 0,C 180,E1 -22404.531,E2 -22404.531} C_VEL
LIN {X 0,Y 185.179,Z 297.185,A -85,B 0,C 180,E1 -22407.822,E2 -22407.822} C_VEL
LIN {X 0,Y 185.537,Z 293.937,A -85,B 0,C 180,E1 -22409.997,E2 -22409.997} C_VEL
LIN {X 0,Y 185.618,Z 287.701,A -85,B 0,C 180,E1 -22413.252,E2 -22413.252} C_VEL
LIN {X 0,Y 185.646,Z 283.623,A -85,B 0,C 180,E1 -22415.002,E2 -22415.002} C_VEL
LIN {X 0,Y 185.031,Z 279.812,A -85,B 0,C 180,E1 -22416.358,E2 -22416.358} C_VEL
LIN {X 0,Y 183.56,Z 275.64,A -85,B 0,C 180,E1 -22417.591,E2 -22417.591} C_VEL
LIN {X 0,Y 179.795,Z 265.041,A -85,B 0,C 180,E1 -22420.233,E2 -22420.233} C_VEL
LIN {X 0,Y 179.354,Z 260.229,A -85,B 0,C 180,E1 -22421.37,E2 -22421.37} C_VEL
LIN {X 0,Y 179.809,Z 249.995,A -85,B 0,C 180,E1 -22423.559,E2 -22423.559} C_VEL
LIN {X 0,Y 180.03,Z 245.299,A -85,B 0,C 180,E1 -22424.407,E2 -22424.407} C_VEL
LIN {X 0,Y 178.753,Z 232.983,A -85,B 0,C 180,E1 -22426.118,E2 -22426.118} C_VEL
LIN {X 0,Y 178.083,Z 219.758,A -85,B 0,C 180,E1 -22427.509,E2 -22427.509} C_VEL
LIN {X 0,Y 180.452,Z 205.703,A -85,B 0,C 180,E1 -22437.859,E2 -22437.859} C_VEL
LIN {X 0,Y 181.157,Z 202.357,A -85,B 0,C 180,E1 -22440.283,E2 -22440.283} C_VEL
LIN {X 0,Y 179.854,Z 196.251,A -85,B 0,C 180,E1 -22444.855,E2 -22444.855} C_VEL
LIN {X 0,Y 178.67,Z 190.224,A -85,B 0,C 180,E1 -22449.544,E2 -22449.544} C_VEL
LIN {X 0,Y 178.455,Z 190.253,A -85,B 0,C 180,E1 -22455.138,E2 -22455.138} C_VEL
LIN {X 0,Y 178.493,Z 190.249,A -85,B 0,C 180,E1 -22458.421,E2 -22458.421} C_VEL
LIN {X 0,Y 178.45,Z 190.255,A -85,B 0,C 180,E1 -22463.789,E2 -22463.789} C_VEL
LIN {X 0,Y 178.48,Z 190.25,A -85,B 0,C 180,E1 -22466.545,E2 -22466.545} C_VEL
LIN {X 0,Y 178.511,Z 190.25,A -85,B 0,C 180,E1 -22470.005,E2 -22470.005} C_VEL
LIN {X 0,Y 178.509,Z 190.244,A -85,B 0,C 180,E1 -22474.884,E2 -22474.884} C_VEL
LIN {X 0,Y 178.611,Z 190.234,A -85,B 0,C 180,E1 -22480.783,E2 -22480.783} C_VEL
LIN {X 0,Y 178.669,Z 190.228,A -85,B 0,C 180,E1 -22486.349,E2 -22486.349} C_VEL
LIN {X 0,Y 178.947,Z 190.191,A -85,B 0,C 180,E1 -22490.961,E2 -22490.961} C_VEL
LIN {X 0,Y 179.144,Z 190.168,A -85,B 0,C 180,E1 -22497.751,E2 -22497.751} C_VEL
LIN {X 0,Y 179.357,Z 190.137,A -85,B 0,C 180,E1 -22500,E2 -22500} C_VEL
LIN {X 0,Y 178.858,Z 190.206,A -85,B 0,C 180,E1 -22504.507,E2 -22504.507} C_VEL
LIN {X 0,Y 178.947,Z 190.191,A -85,B 0,C 180,E1 -22509.038,E2 -22509.038} C_VEL
LIN {X 0,Y 178.669,Z 190.228,A -85,B 0,C 180,E1 -22513.651,E2 -22513.651} C_VEL
LIN {X 0,Y 178.61,Z 190.234,A -85,B 0,C 180,E1 -22519.216,E2 -22519.216} C_VEL
LIN {X 0,Y 178.504,Z 190.244,A -85,B 0,C 180,E1 -22525.113,E2 -22525.113} C_VEL
LIN {X 0,Y 178.449,Z 190.255,A -85,B 0,C 180,E1 -22530.796,E2 -22530.796} C_VEL
LIN {X 0,Y 178.483,Z 190.248,A -85,B 0,C 180,E1 -22534.226,E2 -22534.226} C_VEL
LIN {X 0,Y 178.413,Z 190.26,A -85,B 0,C 180,E1 -22539.07,E2 -22539.07} C_VEL
LIN {X 0,Y 178.413,Z 190.256,A -85,B 0,C 180,E1 -22542.041,E2 -22542.041} C_VEL
LIN {X 0,Y 178.409,Z 190.26,A -85,B 0,C 180,E1 -22545.159,E2 -22545.159} C_VEL
LIN {X 0,Y 178.401,Z 190.261,A -85,B 0,C 180,E1 -22548.46,E2 -22548.46} C_VEL
LIN {X 0,Y 178.416,Z 190.259,A -85,B 0,C 180,E1 -22553.786,E2 -22553.786} C_VEL
LIN {X 0,Y 178.481,Z 190.252,A -85,B 0,C 180,E1 -22556.55,E2 -22556.55} C_VEL
LIN {X 0,Y 178.518,Z 190.241,A -85,B 0,C 180,E1 -22560.01,E2 -22560.01} C_VEL
LIN {X 0,Y 178.53,Z 190.247,A -85,B 0,C 180,E1 -22564.879,E2 -22564.879} C_VEL
LIN {X 0,Y 178.636,Z 190.233,A -85,B 0,C 180,E1 -22570.773,E2 -22570.773} C_VEL
LIN {X 0,Y 178.666,Z 190.226,A -85,B 0,C 180,E1 -22576.352,E2 -22576.352} C_VEL
LIN {X 0,Y 178.978,Z 190.19,A -85,B 0,C 180,E1 -22580.967,E2 -22580.967} C_VEL
LIN {X 0,Y 179.155,Z 190.166,A -85,B 0,C 180,E1 -22587.755,E2 -22587.755} C_VEL
LIN {X 0,Y 179.352,Z 190.146,A -85,B 0,C 180,E1 -22590.004,E2 -22590.004} C_VEL
LIN {X 0,Y 178.874,Z 190.199,A -85,B 0,C 180,E1 -22594.51,E2 -22594.51} C_VEL
LIN {X 0,Y 178.981,Z 190.189,A -85,B 0,C 180,E1 -22599.04,E2 -22599.04} C_VEL
LIN {X 0,Y 178.67,Z 190.226,A -85,B 0,C 180,E1 -22603.655,E2 -22603.655} C_VEL
LIN {X 0,Y 178.623,Z 190.235,A -85,B 0,C 180,E1 -22609.215,E2 -22609.215} C_VEL
LIN {X 0,Y 178.47,Z 190.255,A -85,B 0,C 180,E1 -22615.079,E2 -22615.079} C_VEL
LIN {X 0,Y 178.465,Z 190.25,A -85,B 0,C 180,E1 -22620.797,E2 -22620.797} C_VEL
LIN {X 0,Y 178.488,Z 190.251,A -85,B 0,C 180,E1 -22624.221,E2 -22624.221} C_VEL
LIN {X 0,Y 178.394,Z 190.26,A -85,B 0,C 180,E1 -22629.079,E2 -22629.079} C_VEL
LIN {X 0,Y 178.4,Z 190.262,A -85,B 0,C 180,E1 -22632.049,E2 -22632.049} C_VEL
LIN {X 0,Y 178.4,Z 190.26,A -85,B 0,C 180,E1 -22635.166,E2 -22635.166} C_VEL
LIN {X 0,Y 178.488,Z 190.251,A -85,B 0,C 180,E1 -22640.95,E2 -22640.95} C_VEL
LIN {X 0,Y 178.918,Z 190.289,A -85,B 0,C 180,E1 -22645.264,E2 -22645.264} C_VEL
LIN {X 0,Y 179.459,Z 193.386,A -85,B 0,C 180,E1 -22648.083,E2 -22648.083} C_VEL
LIN {X 0,Y 178.714,Z 197.678,A -85,B 0,C 180,E1 -22651.842,E2 -22651.842} C_VEL
LIN {X 0,Y 177.788,Z 203.28,A -85,B 0,C 180,E1 -22656.715,E2 -22656.715} C_VEL
LIN {X 0,Y 176.97,Z 209.805,A -85,B 0,C 180,E1 -22662.394,E2 -22662.394} C_VEL
LIN {X 0,Y 177.004,Z 217.669,A -85,B 0,C 180,E1 -22669.201,E2 -22669.201} C_VEL
LIN {X 0,Y 177.846,Z 230.364,A -85,B 0,C 180,E1 -22670.905,E2 -22670.905} C_VEL
LIN {X 0,Y 178.326,Z 237.404,A -85,B 0,C 180,E1 -22672.072,E2 -22672.072} C_VEL
LIN {X 0,Y 177.901,Z 248.152,A -85,B 0,C 180,E1 -22674.332,E2 -22674.332} C_VEL
LIN {X 0,Y 177.569,Z 258.792,A -85,B 0,C 180,E1 -22677.164,E2 -22677.164} C_VEL
LIN {X 0,Y 177.184,Z 267.203,A -85,B 0,C 180,E1 -22680,E2 -22680} C_VEL
LIN {X 0,Y 177.167,Z 274.135,A -85,B 0,C 180,E1 -22682.842,E2 -22682.842} C_VEL
LIN {X 0,Y 177.798,Z 280.841,A -85,B 0,C 180,E1 -22686.241,E2 -22686.241} C_VEL
LIN {X 0,Y 178.886,Z 285.341,A -85,B 0,C 180,E1 -22689.042,E2 -22689.042} C_VEL
LIN {X 0,Y 180.564,Z 289.53,A -85,B 0,C 180,E1 -22692.361,E2 -22692.361} C_VEL
LIN {X 0,Y 183.127,Z 292.629,A -85,B 0,C 180,E1 -22695.584,E2 -22695.584} C_VEL
LIN {X 0,Y 185.393,Z 294.104,A -85,B 0,C 180,E1 -22697.654,E2 -22697.654} C_VEL
LIN {X 0,Y 187.858,Z 295.113,A -85,B 0,C 180,E1 -22699.676,E2 -22699.676} C_VEL
LIN {X 0,Y 190.72,Z 295.655,A -85,B 0,C 180,E1 -22701.623,E2 -22701.623} C_VEL
LIN {X 0,Y 193.932,Z 295.739,A -85,B 0,C 180,E1 -22703.493,E2 -22703.493} C_VEL
LIN {X 0,Y 197.446,Z 295.356,A -85,B 0,C 180,E1 -22705.286,E2 -22705.286} C_VEL
LIN {X 0,Y 201.194,Z 294.529,A -85,B 0,C 180,E1 -22707.008,E2 -22707.008} C_VEL
LIN {X 0,Y 205.166,Z 293.245,A -85,B 0,C 180,E1 -22708.658,E2 -22708.658} C_VEL
LIN {X 0,Y 208.986,Z 291.634,A -85,B 0,C 180,E1 -22710.294,E2 -22710.294} C_VEL
LIN {X 0,Y 211.628,Z 290.129,A -85,B 0,C 180,E1 -22712.097,E2 -22712.097} C_VEL
LIN {X 0,Y 214.111,Z 288.513,A -85,B 0,C 180,E1 -22713.918,E2 -22713.918} C_VEL
LIN {X 0,Y 216.359,Z 286.929,A -85,B 0,C 180,E1 -22715.782,E2 -22715.782} C_VEL
LIN {X 0,Y 218.175,Z 285.6,A -85,B 0,C 180,E1 -22717.737,E2 -22717.737} C_VEL
LIN {X 0,Y 219.385,Z 284.748,A -85,B 0,C 180,E1 -22719.844,E2 -22719.844} C_VEL
LIN {X 0,Y 220.316,Z 284.549,A -85,B 0,C 180,E1 -22722.8,E2 -22722.8} C_VEL
LIN {X 0,Y 220.705,Z 285.253,A -85,B 0,C 180,E1 -22725.525,E2 -22725.525} C_VEL
LIN {X 0,Y 220.856,Z 286.569,A -85,B 0,C 180,E1 -22728.064,E2 -22728.064} C_VEL
LIN {X 0,Y 220.138,Z 288.59,A -85,B 0,C 180,E1 -22730.316,E2 -22730.316} C_VEL
LIN {X 0,Y 218.099,Z 290.307,A -85,B 0,C 180,E1 -22731.067,E2 -22731.067} C_VEL
LIN {X 0,Y 211.16,Z 295.196,A -85,B 0,C 180,E1 -22733.192,E2 -22733.192} C_VEL
LIN {X 0,Y 202.689,Z 300.286,A -85,B 0,C 180,E1 -22736.301,E2 -22736.301} C_VEL
LIN {X 0,Y 195.206,Z 303.844,A -85,B 0,C 180,E1 -22739.729,E2 -22739.729} C_VEL
LIN {X 0,Y 191.868,Z 305.127,A -85,B 0,C 180,E1 -22741.56,E2 -22741.56} C_VEL
LIN {X 0,Y 186.468,Z 306.69,A -85,B 0,C 180,E1 -22745.503,E2 -22745.503} C_VEL
LIN {X 0,Y 182.087,Z 306.976,A -85,B 0,C 180,E1 -22749.67,E2 -22749.67} C_VEL
LIN {X 0,Y 179.097,Z 306.024,A -85,B 0,C 180,E1 -22754.053,E2 -22754.053} C_VEL
LIN {X 0,Y 177.635,Z 303.79,A -85,B 0,C 180,E1 -22758.587,E2 -22758.587} C_VEL
LIN {X 0,Y 177.515,Z 300.235,A -85,B 0,C 180,E1 -22763.175,E2 -22763.175} C_VEL
LIN {X 0,Y 178.415,Z 295.026,A -85,B 0,C 180,E1 -22767.739,E2 -22767.739} C_VEL
LIN {X 0,Y 178.786,Z 290.589,A -85,B 0,C 180,E1 -22770.56,E2 -22770.56} C_VEL
LIN {X 0,Y 178.885,Z 283.652,A -85,B 0,C 180,E1 -22773.939,E2 -22773.939} C_VEL
LIN {X 0,Y 178.788,Z 276.234,A -85,B 0,C 180,E1 -22776.769,E2 -22776.769} C_VEL
LIN {X 0,Y 179.051,Z 267.302,A -85,B 0,C 180,E1 -22779.545,E2 -22779.545} C_VEL
LIN {X 0,Y 179.354,Z 260.229,A -85,B 0,C 180,E1 -22781.37,E2 -22781.37} C_VEL
LIN {X 0,Y 178.862,Z 255.378,A -85,B 0,C 180,E1 -22782.407,E2 -22782.407} C_VEL
LIN {X 0,Y 177.346,Z 250.333,A -85,B 0,C 180,E1 -22783.286,E2 -22783.286} C_VEL
LIN {X 0,Y 173.372,Z 239.878,A -85,B 0,C 180,E1 -22784.765,E2 -22784.765} C_VEL
LIN {X 0,Y 171.986,Z 234.325,A -85,B 0,C 180,E1 -22785.476,E2 -22785.476} C_VEL
LIN {X 0,Y 171.753,Z 232.397,A -85,B 0,C 180,E1 -22785.722,E2 -22785.722} C_VEL
LIN {X 0,Y 171.091,Z 219.727,A -85,B 0,C 180,E1 -22787.144,E2 -22787.144} C_VEL
LIN {X 0,Y 171.598,Z 212.293,A -85,B 0,C 180,E1 -22792.893,E2 -22792.893} C_VEL
LIN {X 0,Y 173.774,Z 204.295,A -85,B 0,C 180,E1 -22799.029,E2 -22799.029} C_VEL
LIN {X 0,Y 174.061,Z 202.61,A -85,B 0,C 180,E1 -22800.307,E2 -22800.307} C_VEL
LIN {X 0,Y 172.809,Z 197.003,A -85,B 0,C 180,E1 -22804.701,E2 -22804.701} C_VEL
LIN {X 0,Y 171.623,Z 191.101,A -85,B 0,C 180,E1 -22809.597,E2 -22809.597} C_VEL
LIN {X 0,Y 171.379,Z 191.134,A -85,B 0,C 180,E1 -22815.801,E2 -22815.801} C_VEL
LIN {X 0,Y 171.418,Z 191.131,A -85,B 0,C 180,E1 -22821.161,E2 -22821.161} C_VEL
LIN {X 0,Y 171.396,Z 191.13,A -85,B 0,C 180,E1 -22825.086,E2 -22825.086} C_VEL
LIN {X 0,Y 171.437,Z 191.129,A -85,B 0,C 180,E1 -22830.532,E2 -22830.532} C_VEL
LIN {X 0,Y 171.434,Z 191.128,A -85,B 0,C 180,E1 -22835.798,E2 -22835.798} C_VEL
LIN {X 0,Y 171.567,Z 191.112,A -85,B 0,C 180,E1 -22840.87,E2 -22840.87} C_VEL
LIN {X 0,Y 171.582,Z 191.112,A -85,B 0,C 180,E1 -22845.773,E2 -22845.773} C_VEL
LIN {X 0,Y 171.876,Z 191.071,A -85,B 0,C 180,E1 -22850.586,E2 -22850.586} C_VEL
LIN {X 0,Y 171.813,Z 191.084,A -85,B 0,C 180,E1 -22855.307,E2 -22855.307} C_VEL
LIN {X 0,Y 172.32,Z 191.013,A -85,B 0,C 180,E1 -22860,E2 -22860} C_VEL
LIN {X 0,Y 171.807,Z 191.085,A -85,B 0,C 180,E1 -22864.693,E2 -22864.693} C_VEL
LIN {X 0,Y 171.876,Z 191.071,A -85,B 0,C 180,E1 -22869.413,E2 -22869.413} C_VEL
LIN {X 0,Y 171.582,Z 191.112,A -85,B 0,C 180,E1 -22874.227,E2 -22874.227} C_VEL
LIN {X 0,Y 171.53,Z 191.116,A -85,B 0,C 180,E1 -22879.56,E2 -22879.56} C_VEL
LIN {X 0,Y 171.432,Z 191.126,A -85,B 0,C 180,E1 -22885.6,E2 -22885.6} C_VEL
LIN {X 0,Y 171.406,Z 191.133,A -85,B 0,C 180,E1 -22890.575,E2 -22890.575} C_VEL
LIN {X 0,Y 171.394,Z 191.13,A -85,B 0,C 180,E1 -22895.034,E2 -22895.034} C_VEL
LIN {X 0,Y 171.373,Z 191.137,A -85,B 0,C 180,E1 -22898.821,E2 -22898.821} C_VEL
LIN {X 0,Y 171.334,Z 191.14,A -85,B 0,C 180,E1 -22904.213,E2 -22904.213} C_VEL
LIN {X 0,Y 171.331,Z 191.143,A -85,B 0,C 180,E1 -22908.986,E2 -22908.986} C_VEL
LIN {X 0,Y 171.379,Z 191.132,A -85,B 0,C 180,E1 -22912.044,E2 -22912.044} C_VEL
LIN {X 0,Y 171.392,Z 191.136,A -85,B 0,C 180,E1 -22915.096,E2 -22915.096} C_VEL
LIN {X 0,Y 171.444,Z 191.123,A -85,B 0,C 180,E1 -22920.538,E2 -22920.538} C_VEL
LIN {X 0,Y 171.455,Z 191.126,A -85,B 0,C 180,E1 -22925.806,E2 -22925.806} C_VEL
LIN {X 0,Y 171.593,Z 191.111,A -85,B 0,C 180,E1 -22930.877,E2 -22930.877} C_VEL
LIN {X 0,Y 171.584,Z 191.109,A -85,B 0,C 180,E1 -22935.777,E2 -22935.777} C_VEL
LIN {X 0,Y 171.904,Z 191.072,A -85,B 0,C 180,E1 -22940.592,E2 -22940.592} C_VEL
LIN {X 0,Y 171.826,Z 191.076,A -85,B 0,C 180,E1 -22945.312,E2 -22945.312} C_VEL
LIN {X 0,Y 172.317,Z 191.022,A -85,B 0,C 180,E1 -22950.004,E2 -22950.004} C_VEL
LIN {X 0,Y 171.824,Z 191.076,A -85,B 0,C 180,E1 -22954.696,E2 -22954.696} C_VEL
LIN {X 0,Y 171.907,Z 191.072,A -85,B 0,C 180,E1 -22959.415,E2 -22959.415} C_VEL
LIN {X 0,Y 171.586,Z 191.108,A -85,B 0,C 180,E1 -22964.23,E2 -22964.23} C_VEL
LIN {X 0,Y 171.54,Z 191.115,A -85,B 0,C 180,E1 -22969.557,E2 -22969.557} C_VEL
LIN {X 0,Y 171.407,Z 191.134,A -85,B 0,C 180,E1 -22975.573,E2 -22975.573} C_VEL
LIN {X 0,Y 171.422,Z 191.126,A -85,B 0,C 180,E1 -22980.575,E2 -22980.575} C_VEL
LIN {X 0,Y 171.398,Z 191.135,A -85,B 0,C 180,E1 -22985.038,E2 -22985.038} C_VEL
LIN {X 0,Y 171.35,Z 191.137,A -85,B 0,C 180,E1 -22988.804,E2 -22988.804} C_VEL
LIN {X 0,Y 171.326,Z 191.144,A -85,B 0,C 180,E1 -22994.22,E2 -22994.22} C_VEL
LIN {X 0,Y 171.367,Z 191.137,A -85,B 0,C 180,E1 -22998.991,E2 -22998.991} C_VEL
LIN {X 0,Y 171.879,Z 191.105,A -85,B 0,C 180,E1 -23005.435,E2 -23005.435} C_VEL
LIN {X 0,Y 172.361,Z 193.826,A -85,B 0,C 180,E1 -23007.99,E2 -23007.99} C_VEL
LIN {X 0,Y 171.6,Z 198.125,A -85,B 0,C 180,E1 -23011.901,E2 -23011.901} C_VEL
LIN {X 0,Y 170.653,Z 203.744,A -85,B 0,C 180,E1 -23016.969,E2 -23016.969} C_VEL
LIN {X 0,Y 169.809,Z 210.566,A -85,B 0,C 180,E1 -23023.159,E2 -23023.159} C_VEL
LIN {X 0,Y 170.053,Z 217.921,A -85,B 0,C 180,E1 -23029.658,E2 -23029.658} C_VEL
LIN {X 0,Y 170.899,Z 230.147,A -85,B 0,C 180,E1 -23031.352,E2 -23031.352} C_VEL
LIN {X 0,Y 171.386,Z 236.416,A -85,B 0,C 180,E1 -23032.415,E2 -23032.415} C_VEL
LIN {X 0,Y 170.986,Z 247.052,A -85,B 0,C 180,E1 -23034.694,E2 -23034.694} C_VEL
LIN {X 0,Y 170.68,Z 257.865,A -85,B 0,C 180,E1 -23037.64,E2 -23037.64} C_VEL
LIN {X 0,Y 170.317,Z 266.452,A -85,B 0,C 180,E1 -23040.591,E2 -23040.591} C_VEL
LIN {X 0,Y 170.417,Z 274.752,A -85,B 0,C 180,E1 -23044.139,E2 -23044.139} C_VEL
LIN {X 0,Y 171.046,Z 280.342,A -85,B 0,C 180,E1 -23047.081,E2 -23047.081} C_VEL
LIN {X 0,Y 172.445,Z 285.799,A -85,B 0,C 180,E1 -23050.568,E2 -23050.568} C_VEL
LIN {X 0,Y 174.484,Z 289.985,A -85,B 0,C 180,E1 -23053.985,E2 -23053.985} C_VEL
LIN {X 0,Y 176.32,Z 292.19,A -85,B 0,C 180,E1 -23056.202,E2 -23056.202} C_VEL
LIN {X 0,Y 178.647,Z 293.903,A -85,B 0,C 180,E1 -23058.344,E2 -23058.344} C_VEL
LIN {X 0,Y 181.208,Z 295.186,A -85,B 0,C 180,E1 -23060.43,E2 -23060.43} C_VEL
LIN {X 0,Y 184.137,Z 295.99,A -85,B 0,C 180,E1 -23062.438,E2 -23062.438} C_VEL
LIN {X 0,Y 187.451,Z 296.366,A -85,B 0,C 180,E1 -23064.357,E2 -23064.357} C_VEL
LIN {X 0,Y 191.07,Z 296.262,A -85,B 0,C 180,E1 -23066.193,E2 -23066.193} C_VEL
LIN {X 0,Y 194.941,Z 295.735,A -85,B 0,C 180,E1 -23067.949,E2 -23067.949} C_VEL
LIN {X 0,Y 199.06,Z 294.751,A -85,B 0,C 180,E1 -23069.623,E2 -23069.623} C_VEL
LIN {X 0,Y 203.047,Z 293.436,A -85,B 0,C 180,E1 -23071.278,E2 -23071.278} C_VEL
LIN {X 0,Y 205.848,Z 292.205,A -85,B 0,C 180,E1 -23073.112,E2 -23073.112} C_VEL
LIN {X 0,Y 208.474,Z 290.875,A -85,B 0,C 180,E1 -23074.967,E2 -23074.967} C_VEL
LIN {X 0,Y 210.786,Z 289.612,A -85,B 0,C 180,E1 -23076.881,E2 -23076.881} C_VEL
LIN {X 0,Y 212.537,Z 288.651,A -85,B 0,C 180,E1 -23078.923,E2 -23078.923} C_VEL
LIN {X 0,Y 213.655,Z 288.194,A -85,B 0,C 180,E1 -23081.139,E2 -23081.139} C_VEL
LIN {X 0,Y 214.351,Z 288.397,A -85,B 0,C 180,E1 -23083.833,E2 -23083.833} C_VEL
LIN {X 0,Y 214.64,Z 289.307,A -85,B 0,C 180,E1 -23086.556,E2 -23086.556} C_VEL
LIN {X 0,Y 214.284,Z 290.857,A -85,B 0,C 180,E1 -23089.005,E2 -23089.005} C_VEL
LIN {X 0,Y 212.74,Z 292.18,A -85,B 0,C 180,E1 -23089.891,E2 -23089.891} C_VEL
LIN {X 0,Y 204.023,Z 297.463,A -85,B 0,C 180,E1 -23092.546,E2 -23092.546} C_VEL
LIN {X 0,Y 196.862,Z 301.066,A -85,B 0,C 180,E1 -23095.162,E2 -23095.162} C_VEL
LIN {X 0,Y 189.119,Z 304.101,A -85,B 0,C 180,E1 -23098.646,E2 -23098.646} C_VEL
LIN {X 0,Y 185.401,Z 305.212,A -85,B 0,C 180,E1 -23100.676,E2 -23100.676} C_VEL
LIN {X 0,Y 180.04,Z 306.269,A -85,B 0,C 180,E1 -23104.567,E2 -23104.567} C_VEL
LIN {X 0,Y 175.486,Z 306.122,A -85,B 0,C 180,E1 -23108.869,E2 -23108.869} C_VEL
LIN {X 0,Y 172.37,Z 304.788,A -85,B 0,C 180,E1 -23113.413,E2 -23113.413} C_VEL
LIN {X 0,Y 170.837,Z 302.201,A -85,B 0,C 180,E1 -23118.126,E2 -23118.126} C_VEL
LIN {X 0,Y 170.725,Z 298.278,A -85,B 0,C 180,E1 -23122.902,E2 -23122.902} C_VEL
LIN {X 0,Y 171.338,Z 294.27,A -85,B 0,C 180,E1 -23126.469,E2 -23126.469} C_VEL
LIN {X 0,Y 171.933,Z 290.999,A -85,B 0,C 180,E1 -23128.825,E2 -23128.825} C_VEL
LIN {X 0,Y 172.065,Z 285.704,A -85,B 0,C 180,E1 -23131.752,E2 -23131.752} C_VEL
LIN {X 0,Y 172.094,Z 279.091,A -85,B 0,C 180,E1 -23134.681,E2 -23134.681} C_VEL
LIN {X 0,Y 172.104,Z 270.804,A -85,B 0,C 180,E1 -23137.623,E2 -23137.623} C_VEL
LIN {X 0,Y 172.366,Z 261.083,A -85,B 0,C 180,E1 -23140.417,E2 -23140.417} C_VEL
LIN {X 0,Y 172.814,Z 250.719,A -85,B 0,C 180,E1 -23142.801,E2 -23142.801} C_VEL
LIN {X 0,Y 173.008,Z 243.762,A -85,B 0,C 180,E1 -23144.103,E2 -23144.103} C_VEL
LIN {X 0,Y 171.753,Z 232.397,A -85,B 0,C 180,E1 -23145.722,E2 -23145.722} C_VEL
LIN {X 0,Y 170.776,Z 228.582,A -85,B 0,C 180,E1 -23146.214,E2 -23146.214} C_VEL
LIN {X 0,Y 167.526,Z 222.844,A -85,B 0,C 180,E1 -23147.098,E2 -23147.098} C_VEL
LIN {X 0,Y 164.99,Z 219.026,A -85,B 0,C 180,E1 -23148.102,E2 -23148.102} C_VEL
LIN {X 0,Y 163.915,Z 216.73,A -85,B 0,C 180,E1 -23149.158,E2 -23149.158} C_VEL
LIN {X 0,Y 163.861,Z 216.148,A -85,B 0,C 180,E1 -23149.57,E2 -23149.57} C_VEL
LIN {X 0,Y 166.091,Z 206.092,A -85,B 0,C 180,E1 -23157.735,E2 -23157.735} C_VEL
LIN {X 0,Y 166.942,Z 202.827,A -85,B 0,C 180,E1 -23160.339,E2 -23160.339} C_VEL
LIN {X 0,Y 165.719,Z 197.44,A -85,B 0,C 180,E1 -23164.737,E2 -23164.737} C_VEL
LIN {X 0,Y 164.598,Z 191.977,A -85,B 0,C 180,E1 -23169.42,E2 -23169.42} C_VEL
LIN {X 0,Y 164.352,Z 192.011,A -85,B 0,C 180,E1 -23173.368,E2 -23173.368} C_VEL
LIN {X 0,Y 164.349,Z 192.007,A -85,B 0,C 180,E1 -23176.827,E2 -23176.827} C_VEL
LIN {X 0,Y 164.362,Z 192.012,A -85,B 0,C 180,E1 -23180.317,E2 -23180.317} C_VEL
LIN {X 0,Y 164.335,Z 192.011,A -85,B 0,C 180,E1 -23184.339,E2 -23184.339} C_VEL
LIN {X 0,Y 164.379,Z 192.008,A -85,B 0,C 180,E1 -23189.132,E2 -23189.132} C_VEL
LIN {X 0,Y 164.395,Z 192.002,A -85,B 0,C 180,E1 -23194.69,E2 -23194.69} C_VEL
LIN {X 0,Y 164.473,Z 191.996,A -85,B 0,C 180,E1 -23200.05,E2 -23200.05} C_VEL
LIN {X 0,Y 164.524,Z 191.989,A -85,B 0,C 180,E1 -23205.149,E2 -23205.149} C_VEL
LIN {X 0,Y 164.797,Z 191.953,A -85,B 0,C 180,E1 -23210.178,E2 -23210.178} C_VEL
LIN {X 0,Y 164.839,Z 191.947,A -85,B 0,C 180,E1 -23212.651,E2 -23212.651} C_VEL
LIN {X 0,Y 165.04,Z 191.925,A -85,B 0,C 180,E1 -23217.559,E2 -23217.559} C_VEL
LIN {X 0,Y 165.282,Z 191.89,A -85,B 0,C 180,E1 -23220,E2 -23220} C_VEL
LIN {X 0,Y 164.757,Z 191.963,A -85,B 0,C 180,E1 -23224.894,E2 -23224.894} C_VEL
LIN {X 0,Y 164.838,Z 191.948,A -85,B 0,C 180,E1 -23227.349,E2 -23227.349} C_VEL
LIN {X 0,Y 164.742,Z 191.963,A -85,B 0,C 180,E1 -23231.152,E2 -23231.152} C_VEL
LIN {X 0,Y 164.473,Z 191.991,A -85,B 0,C 180,E1 -23237.404,E2 -23237.404} C_VEL
LIN {X 0,Y 164.461,Z 191.998,A -85,B 0,C 180,E1 -23239.991,E2 -23239.991} C_VEL
LIN {X 0,Y 164.358,Z 192.007,A -85,B 0,C 180,E1 -23246.119,E2 -23246.119} C_VEL
LIN {X 0,Y 164.346,Z 192.012,A -85,B 0,C 180,E1 -23251.22,E2 -23251.22} C_VEL
LIN {X 0,Y 164.303,Z 192.017,A -85,B 0,C 180,E1 -23256.787,E2 -23256.787} C_VEL
LIN {X 0,Y 164.294,Z 192.019,A -85,B 0,C 180,E1 -23259.915,E2 -23259.915} C_VEL
LIN {X 0,Y 164.298,Z 192.014,A -85,B 0,C 180,E1 -23263.355,E2 -23263.355} C_VEL
LIN {X 0,Y 164.284,Z 192.02,A -85,B 0,C 180,E1 -23266.812,E2 -23266.812} C_VEL
LIN {X 0,Y 164.288,Z 192.016,A -85,B 0,C 180,E1 -23270.355,E2 -23270.355} C_VEL
LIN {X 0,Y 164.323,Z 192.014,A -85,B 0,C 180,E1 -23274.352,E2 -23274.352} C_VEL
LIN {X 0,Y 164.385,Z 192.004,A -85,B 0,C 180,E1 -23279.139,E2 -23279.139} C_VEL
LIN {X 0,Y 164.413,Z 192.006,A -85,B 0,C 180,E1 -23284.698,E2 -23284.698} C_VEL
LIN {X 0,Y 164.483,Z 191.992,A -85,B 0,C 180,E1 -23290.054,E2 -23290.054} C_VEL
LIN {X 0,Y 164.531,Z 191.987,A -85,B 0,C 180,E1 -23295.154,E2 -23295.154} C_VEL
LIN {X 0,Y 164.834,Z 191.952,A -85,B 0,C 180,E1 -23300.184,E2 -23300.184} C_VEL
LIN {X 0,Y 164.861,Z 191.948,A -85,B 0,C 180,E1 -23302.656,E2 -23302.656} C_VEL
LIN {X 0,Y 165.051,Z 191.922,A -85,B 0,C 180,E1 -23307.563,E2 -23307.563} C_VEL
LIN {X 0,Y 165.282,Z 191.898,A -85,B 0,C 180,E1 -23310.004,E2 -23310.004} C_VEL
LIN {X 0,Y 164.774,Z 191.954,A -85,B 0,C 180,E1 -23314.897,E2 -23314.897} C_VEL
LIN {X 0,Y 164.863,Z 191.948,A -85,B 0,C 180,E1 -23317.351,E2 -23317.351} C_VEL
LIN {X 0,Y 164.753,Z 191.961,A -85,B 0,C 180,E1 -23321.149,E2 -23321.149} C_VEL
LIN {X 0,Y 164.486,Z 191.997,A -85,B 0,C 180,E1 -23327.407,E2 -23327.407} C_VEL
LIN {X 0,Y 164.476,Z 191.993,A -85,B 0,C 180,E1 -23329.993,E2 -23329.993} C_VEL
LIN {X 0,Y 164.343,Z 192.013,A -85,B 0,C 180,E1 -23336.098,E2 -23336.098} C_VEL
LIN {X 0,Y 164.362,Z 192.009,A -85,B 0,C 180,E1 -23341.22,E2 -23341.22} C_VEL
LIN {X 0,Y 164.286,Z 192.019,A -85,B 0,C 180,E1 -23346.796,E2 -23346.796} C_VEL
LIN {X 0,Y 164.292,Z 192.016,A -85,B 0,C 180,E1 -23349.92,E2 -23349.92} C_VEL
LIN {X 0,Y 164.286,Z 192.02,A -85,B 0,C 180,E1 -23353.344,E2 -23353.344} C_VEL
LIN {X 0,Y 164.3,Z 192.014,A -85,B 0,C 180,E1 -23356.811,E2 -23356.811} C_VEL
LIN {X 0,Y 164.561,Z 191.984,A -85,B 0,C 180,E1 -23363.28,E2 -23363.28} C_VEL
LIN {X 0,Y 164.888,Z 192.099,A -85,B 0,C 180,E1 -23365.805,E2 -23365.805} C_VEL
LIN {X 0,Y 165.226,Z 194.655,A -85,B 0,C 180,E1 -23368.295,E2 -23368.295} C_VEL
LIN {X 0,Y 164.202,Z 199.82,A -85,B 0,C 180,E1 -23373.168,E2 -23373.168} C_VEL
LIN {X 0,Y 163.298,Z 205.532,A -85,B 0,C 180,E1 -23378.542,E2 -23378.542} C_VEL
LIN {X 0,Y 162.576,Z 212.333,A -85,B 0,C 180,E1 -23384.967,E2 -23384.967} C_VEL
LIN {X 0,Y 163.085,Z 217.816,A -85,B 0,C 180,E1 -23390.121,E2 -23390.121} C_VEL
LIN {X 0,Y 164.068,Z 230.731,A -85,B 0,C 180,E1 -23392.003,E2 -23392.003} C_VEL
LIN {X 0,Y 164.448,Z 236.004,A -85,B 0,C 180,E1 -23392.942,E2 -23392.942} C_VEL
LIN {X 0,Y 164.056,Z 246.955,A -85,B 0,C 180,E1 -23395.393,E2 -23395.393} C_VEL
LIN {X 0,Y 163.83,Z 256.803,A -85,B 0,C 180,E1 -23398.156,E2 -23398.156} C_VEL
LIN {X 0,Y 163.487,Z 265.538,A -85,B 0,C 180,E1 -23401.232,E2 -23401.232} C_VEL
LIN {X 0,Y 163.632,Z 273.991,A -85,B 0,C 180,E1 -23404.928,E2 -23404.928} C_VEL
LIN {X 0,Y 164.598,Z 280.791,A -85,B 0,C 180,E1 -23408.595,E2 -23408.595} C_VEL
LIN {X 0,Y 166.137,Z 286.18,A -85,B 0,C 180,E1 -23412.211,E2 -23412.211} C_VEL
LIN {X 0,Y 168.579,Z 290.391,A -85,B 0,C 180,E1 -23415.723,E2 -23415.723} C_VEL
LIN {X 0,Y 171.932,Z 293.53,A -85,B 0,C 180,E1 -23419.088,E2 -23419.088} C_VEL
LIN {X 0,Y 174.593,Z 295.079,A -85,B 0,C 180,E1 -23421.241,E2 -23421.241} C_VEL
LIN {X 0,Y 177.595,Z 296.146,A -85,B 0,C 180,E1 -23423.312,E2 -23423.312} C_VEL
LIN {X 0,Y 181.019,Z 296.81,A -85,B 0,C 180,E1 -23425.282,E2 -23425.282} C_VEL
LIN {X 0,Y 184.73,Z 296.993,A -85,B 0,C 180,E1 -23427.164,E2 -23427.164} C_VEL
LIN {X 0,Y 188.738,Z 296.766,A -85,B 0,C 180,E1 -23428.952,E2 -23428.952} C_VEL
LIN {X 0,Y 192.967,Z 296.084,A -85,B 0,C 180,E1 -23430.657,E2 -23430.657} C_VEL
LIN {X 0,Y 197.137,Z 295.059,A -85,B 0,C 180,E1 -23432.328,E2 -23432.328} C_VEL
LIN {X 0,Y 200.078,Z 294.105,A -85,B 0,C 180,E1 -23434.196,E2 -23434.196} C_VEL
LIN {X 0,Y 202.809,Z 293.068,A -85,B 0,C 180,E1 -23436.094,E2 -23436.094} C_VEL
LIN {X 0,Y 205.108,Z 292.131,A -85,B 0,C 180,E1 -23438.081,E2 -23438.081} C_VEL
LIN {X 0,Y 206.761,Z 291.524,A -85,B 0,C 180,E1 -23440.228,E2 -23440.228} C_VEL
LIN {X 0,Y 207.693,Z 291.506,A -85,B 0,C 180,E1 -23442.592,E2 -23442.592} C_VEL
LIN {X 0,Y 208.132,Z 292.042,A -85,B 0,C 180,E1 -23445.163,E2 -23445.163} C_VEL
LIN {X 0,Y 207.992,Z 293.333,A -85,B 0,C 180,E1 -23448.02,E2 -23448.02} C_VEL
LIN {X 0,Y 204.969,Z 295.289,A -85,B 0,C 180,E1 -23449.344,E2 -23449.344} C_VEL
LIN {X 0,Y 195.507,Z 299.902,A -85,B 0,C 180,E1 -23452.327,E2 -23452.327} C_VEL
LIN {X 0,Y 187.011,Z 303.111,A -85,B 0,C 180,E1 -23455.684,E2 -23455.684} C_VEL
LIN {X 0,Y 179.527,Z 304.993,A -85,B 0,C 180,E1 -23459.405,E2 -23459.405} C_VEL
LIN {X 0,Y 173.664,Z 305.681,A -85,B 0,C 180,E1 -23463.563,E2 -23463.563} C_VEL
LIN {X 0,Y 168.925,Z 305.115,A -85,B 0,C 180,E1 -23468.007,E2 -23468.007} C_VEL
LIN {X 0,Y 165.684,Z 303.383,A -85,B 0,C 180,E1 -23472.723,E2 -23472.723} C_VEL
LIN {X 0,Y 164.106,Z 300.464,A -85,B 0,C 180,E1 -23477.632,E2 -23477.632} C_VEL
LIN {X 0,Y 164.006,Z 296.169,A -85,B 0,C 180,E1 -23482.61,E2 -23482.61} C_VEL
LIN {X 0,Y 164.682,Z 291.883,A -85,B 0,C 180,E1 -23486.326,E2 -23486.326} C_VEL
LIN {X 0,Y 165.262,Z 288.375,A -85,B 0,C 180,E1 -23488.778,E2 -23488.778} C_VEL
LIN {X 0,Y 165.378,Z 282.721,A -85,B 0,C 180,E1 -23491.823,E2 -23491.823} C_VEL
LIN {X 0,Y 165.358,Z 275.608,A -85,B 0,C 180,E1 -23494.872,E2 -23494.872} C_VEL
LIN {X 0,Y 165.399,Z 265.713,A -85,B 0,C 180,E1 -23498.241,E2 -23498.241} C_VEL
LIN {X 0,Y 165.695,Z 256.733,A -85,B 0,C 180,E1 -23500.705,E2 -23500.705} C_VEL
LIN {X 0,Y 166.156,Z 245.472,A -85,B 0,C 180,E1 -23503.167,E2 -23503.167} C_VEL
LIN {X 0,Y 165.138,Z 235.214,A -85,B 0,C 180,E1 -23504.79,E2 -23504.79} C_VEL
LIN {X 0,Y 164.191,Z 222.02,A -85,B 0,C 180,E1 -23506.39,E2 -23506.39} C_VEL
LIN {X 0,Y 164.147,Z 219.749,A -85,B 0,C 180,E1 -23506.634,E2 -23506.634} C_VEL
LIN {X 0,Y 163.861,Z 216.148,A -85,B 0,C 180,E1 -23509.57,E2 -23509.57} C_VEL
LIN {X 0,Y 163.521,Z 213.813,A -85,B 0,C 180,E1 -23511.464,E2 -23511.464} C_VEL
LIN {X 0,Y 159.555,Z 205.255,A -85,B 0,C 180,E1 -23518.466,E2 -23518.466} C_VEL
LIN {X 0,Y 159.653,Z 203.688,A -85,B 0,C 180,E1 -23519.776,E2 -23519.776} C_VEL
LIN {X 0,Y 159.839,Z 202.976,A -85,B 0,C 180,E1 -23520.369,E2 -23520.369} C_VEL
LIN {X 0,Y 158.496,Z 197.351,A -85,B 0,C 180,E1 -23525.195,E2 -23525.195} C_VEL
LIN {X 0,Y 157.571,Z 192.852,A -85,B 0,C 180,E1 -23529.362,E2 -23529.362} C_VEL
LIN {X 0,Y 157.238,Z 192.896,A -85,B 0,C 180,E1 -23535.649,E2 -23535.649} C_VEL
LIN {X 0,Y 157.278,Z 192.893,A -85,B 0,C 180,E1 -23541.274,E2 -23541.274} C_VEL
LIN {X 0,Y 157.282,Z 192.889,A -85,B 0,C 180,E1 -23544.486,E2 -23544.486} C_VEL
LIN {X 0,Y 157.283,Z 192.892,A -85,B 0,C 180,E1 -23548.093,E2 -23548.093} C_VEL
LIN {X 0,Y 157.304,Z 192.887,A -85,B 0,C 180,E1 -23553.462,E2 -23553.462} C_VEL
LIN {X 0,Y 157.381,Z 192.881,A -85,B 0,C 180,E1 -23559.667,E2 -23559.667} C_VEL
LIN {X 0,Y 157.45,Z 192.869,A -85,B 0,C 180,E1 -23564.465,E2 -23564.465} C_VEL
LIN {X 0,Y 157.723,Z 192.835,A -85,B 0,C 180,E1 -23569.733,E2 -23569.733} C_VEL
LIN {X 0,Y 157.797,Z 192.824,A -85,B 0,C 180,E1 -23572.321,E2 -23572.321} C_VEL
LIN {X 0,Y 158.245,Z 192.766,A -85,B 0,C 180,E1 -23580,E2 -23580} C_VEL
LIN {X 0,Y 157.796,Z 192.824,A -85,B 0,C 180,E1 -23587.678,E2 -23587.678} C_VEL
LIN {X 0,Y 157.671,Z 192.844,A -85,B 0,C 180,E1 -23591.321,E2 -23591.321} C_VEL
LIN {X 0,Y 157.45,Z 192.869,A -85,B 0,C 180,E1 -23595.534,E2 -23595.534} C_VEL
LIN {X 0,Y 157.355,Z 192.883,A -85,B 0,C 180,E1 -23600.935,E2 -23600.935} C_VEL
LIN {X 0,Y 157.298,Z 192.888,A -85,B 0,C 180,E1 -23606.683,E2 -23606.683} C_VEL
LIN {X 0,Y 157.259,Z 192.893,A -85,B 0,C 180,E1 -23612.431,E2 -23612.431} C_VEL
LIN {X 0,Y 157.272,Z 192.893,A -85,B 0,C 180,E1 -23616.459,E2 -23616.459} C_VEL
LIN {X 0,Y 157.205,Z 192.897,A -85,B 0,C 180,E1 -23622.113,E2 -23622.113} C_VEL
LIN {X 0,Y 157.203,Z 192.902,A -85,B 0,C 180,E1 -23627.893,E2 -23627.893} C_VEL
LIN {X 0,Y 157.261,Z 192.895,A -85,B 0,C 180,E1 -23633.554,E2 -23633.554} C_VEL
LIN {X 0,Y 157.288,Z 192.89,A -85,B 0,C 180,E1 -23638.099,E2 -23638.099} C_VEL
LIN {X 0,Y 157.318,Z 192.888,A -85,B 0,C 180,E1 -23643.47,E2 -23643.47} C_VEL
LIN {X 0,Y 157.392,Z 192.875,A -85,B 0,C 180,E1 -23649.67,E2 -23649.67} C_VEL
LIN {X 0,Y 157.462,Z 192.871,A -85,B 0,C 180,E1 -23654.471,E2 -23654.471} C_VEL
LIN {X 0,Y 157.748,Z 192.833,A -85,B 0,C 180,E1 -23659.739,E2 -23659.739} C_VEL
LIN {X 0,Y 157.821,Z 192.826,A -85,B 0,C 180,E1 -23662.327,E2 -23662.327} C_VEL
LIN {X 0,Y 158.246,Z 192.775,A -85,B 0,C 180,E1 -23670.004,E2 -23670.004} C_VEL
LIN {X 0,Y 157.823,Z 192.826,A -85,B 0,C 180,E1 -23677.681,E2 -23677.681} C_VEL
LIN {X 0,Y 157.682,Z 192.842,A -85,B 0,C 180,E1 -23681.318,E2 -23681.318} C_VEL
LIN {X 0,Y 157.459,Z 192.871,A -85,B 0,C 180,E1 -23685.538,E2 -23685.538} C_VEL
LIN {X 0,Y 157.365,Z 192.879,A -85,B 0,C 180,E1 -23690.937,E2 -23690.937} C_VEL
LIN {X 0,Y 157.271,Z 192.894,A -85,B 0,C 180,E1 -23696.652,E2 -23696.652} C_VEL
LIN {X 0,Y 157.273,Z 192.892,A -85,B 0,C 180,E1 -23702.432,E2 -23702.432} C_VEL
LIN {X 0,Y 157.264,Z 192.895,A -85,B 0,C 180,E1 -23706.447,E2 -23706.447} C_VEL
LIN {X 0,Y 157.196,Z 192.903,A -85,B 0,C 180,E1 -23712.12,E2 -23712.12} C_VEL
LIN {X 0,Y 157.23,Z 192.894,A -85,B 0,C 180,E1 -23717.896,E2 -23717.896} C_VEL
LIN {X 0,Y 157.658,Z 192.844,A -85,B 0,C 180,E1 -23724.584,E2 -23724.584} C_VEL
LIN {X 0,Y 157.892,Z 193.053,A -85,B 0,C 180,E1 -23726.195,E2 -23726.195} C_VEL
LIN {X 0,Y 158.092,Z 194.6,A -85,B 0,C 180,E1 -23727.761,E2 -23727.761} C_VEL
LIN {X 0,Y 157.668,Z 197.506,A -85,B 0,C 180,E1 -23730.638,E2 -23730.638} C_VEL
LIN {X 0,Y 156.573,Z 203.136,A -85,B 0,C 180,E1 -23736.173,E2 -23736.173} C_VEL
LIN {X 0,Y 155.639,Z 209.986,A -85,B 0,C 180,E1 -23742.932,E2 -23742.932} C_VEL
LIN {X 0,Y 156.185,Z 217.976,A -85,B 0,C 180,E1 -23750.719,E2 -23750.719} C_VEL
LIN {X 0,Y 157.18,Z 230.559,A -85,B 0,C 180,E1 -23752.614,E2 -23752.614} C_VEL
LIN {X 0,Y 157.527,Z 235.814,A -85,B 0,C 180,E1 -23753.596,E2 -23753.596} C_VEL
LIN {X 0,Y 157.163,Z 246.71,A -85,B 0,C 180,E1 -23756.154,E2 -23756.154} C_VEL
LIN {X 0,Y 157.025,Z 255.601,A -85,B 0,C 180,E1 -23758.718,E2 -23758.718} C_VEL
LIN {X 0,Y 156.704,Z 264.499,A -85,B 0,C 180,E1 -23761.928,E2 -23761.928} C_VEL
LIN {X 0,Y 156.915,Z 273.145,A -85,B 0,C 180,E1 -23765.784,E2 -23765.784} C_VEL
LIN {X 0,Y 157.991,Z 280.129,A -85,B 0,C 180,E1 -23769.603,E2 -23769.603} C_VEL
LIN {X 0,Y 159.345,Z 284.859,A -85,B 0,C 180,E1 -23772.74,E2 -23772.74} C_VEL
LIN {X 0,Y 161.81,Z 289.441,A -85,B 0,C 180,E1 -23776.399,E2 -23776.399} C_VEL
LIN {X 0,Y 165.272,Z 292.976,A -85,B 0,C 180,E1 -23779.889,E2 -23779.889} C_VEL
LIN {X 0,Y 168.018,Z 294.779,A -85,B 0,C 180,E1 -23782.115,E2 -23782.115} C_VEL
LIN {X 0,Y 171.102,Z 296.117,A -85,B 0,C 180,E1 -23784.252,E2 -23784.252} C_VEL
LIN {X 0,Y 174.622,Z 297.064,A -85,B 0,C 180,E1 -23786.278,E2 -23786.278} C_VEL
LIN {X 0,Y 178.444,Z 297.536,A -85,B 0,C 180,E1 -23788.205,E2 -23788.205} C_VEL
LIN {X 0,Y 182.573,Z 297.608,A -85,B 0,C 180,E1 -23790.028,E2 -23790.028} C_VEL
LIN {X 0,Y 186.939,Z 297.224,A -85,B 0,C 180,E1 -23791.758,E2 -23791.758} C_VEL
LIN {X 0,Y 191.257,Z 296.503,A -85,B 0,C 180,E1 -23793.449,E2 -23793.449} C_VEL
LIN {X 0,Y 194.321,Z 295.816,A -85,B 0,C 180,E1 -23795.357,E2 -23795.357} C_VEL
LIN {X 0,Y 197.134,Z 295.062,A -85,B 0,C 180,E1 -23797.306,E2 -23797.306} C_VEL
LIN {X 0,Y 199.327,Z 294.465,A -85,B 0,C 180,E1 -23799.395,E2 -23799.395} C_VEL
LIN {X 0,Y 200.83,Z 294.234,A -85,B 0,C 180,E1 -23801.675,E2 -23801.675} C_VEL
LIN {X 0,Y 201.452,Z 294.601,A -85,B 0,C 180,E1 -23804.246,E2 -23804.246} C_VEL
LIN {X 0,Y 201.496,Z 295.579,A -85,B 0,C 180,E1 -23807.093,E2 -23807.093} C_VEL
LIN {X 0,Y 199.688,Z 296.638,A -85,B 0,C 180,E1 -23808.029,E2 -23808.029} C_VEL
LIN {X 0,Y 189.962,Z 300.64,A -85,B 0,C 180,E1 -23811.024,E2 -23811.024} C_VEL
LIN {X 0,Y 181.193,Z 303.304,A -85,B 0,C 180,E1 -23814.418,E2 -23814.418} C_VEL
LIN {X 0,Y 173.464,Z 304.681,A -85,B 0,C 180,E1 -23818.213,E2 -23818.213} C_VEL
LIN {X 0,Y 167.351,Z 304.912,A -85,B 0,C 180,E1 -23822.483,E2 -23822.483} C_VEL
LIN {X 0,Y 162.433,Z 303.942,A -85,B 0,C 180,E1 -23827.079,E2 -23827.079} C_VEL
LIN {X 0,Y 159.074,Z 301.818,A -85,B 0,C 180,E1 -23831.981,E2 -23831.981} C_VEL
LIN {X 0,Y 157.432,Z 298.534,A -85,B 0,C 180,E1 -23837.099,E2 -23837.099} C_VEL
LIN {X 0,Y 157.338,Z 293.867,A -85,B 0,C 180,E1 -23842.295,E2 -23842.295} C_VEL
LIN {X 0,Y 158.095,Z 289.317,A -85,B 0,C 180,E1 -23846.173,E2 -23846.173} C_VEL
LIN {X 0,Y 158.668,Z 285.544,A -85,B 0,C 180,E1 -23848.727,E2 -23848.727} C_VEL
LIN {X 0,Y 158.741,Z 279.491,A -85,B 0,C 180,E1 -23851.899,E2 -23851.899} C_VEL
LIN {X 0,Y 158.671,Z 273.473,A -85,B 0,C 180,E1 -23854.442,E2 -23854.442} C_VEL
LIN {X 0,Y 158.667,Z 264.305,A -85,B 0,C 180,E1 -23857.632,E2 -23857.632} C_VEL
LIN {X 0,Y 158.947,Z 254.053,A -85,B 0,C 180,E1 -23860.487,E2 -23860.487} C_VEL
LIN {X 0,Y 159.321,Z 243.857,A -85,B 0,C 180,E1 -23862.738,E2 -23862.738} C_VEL
LIN {X 0,Y 157.914,Z 231.792,A -85,B 0,C 180,E1 -23864.63,E2 -23864.63} C_VEL
LIN {X 0,Y 157.206,Z 219.671,A -85,B 0,C 180,E1 -23866.137,E2 -23866.137} C_VEL
LIN {X 0,Y 156.826,Z 215.443,A -85,B 0,C 180,E1 -23869.763,E2 -23869.763} C_VEL
LIN {X 0,Y 159.008,Z 205.965,A -85,B 0,C 180,E1 -23877.873,E2 -23877.873} C_VEL
LIN {X 0,Y 159.653,Z 203.688,A -85,B 0,C 180,E1 -23879.776,E2 -23879.776} C_VEL
LIN {X 0,Y 159.303,Z 202.433,A -85,B 0,C 180,E1 -23880.839,E2 -23880.839} C_VEL
LIN {X 0,Y 157.339,Z 200.844,A -85,B 0,C 180,E1 -23882.246,E2 -23882.246} C_VEL
LIN {X 0,Y 152.172,Z 197.873,A -85,B 0,C 180,E1 -23885.062,E2 -23885.062} C_VEL
LIN {X 0,Y 151.08,Z 196.407,A -85,B 0,C 180,E1 -23886.448,E2 -23886.448} C_VEL
LIN {X 0,Y 150.523,Z 193.73,A -85,B 0,C 180,E1 -23889.14,E2 -23889.14} C_VEL
LIN {X 0,Y 150.189,Z 193.774,A -85,B 0,C 180,E1 -23895.419,E2 -23895.419} C_VEL
LIN {X 0,Y 150.213,Z 193.772,A -85,B 0,C 180,E1 -23899.079,E2 -23899.079} C_VEL
LIN {X 0,Y 150.227,Z 193.771,A -85,B 0,C 180,E1 -23902.676,E2 -23902.676} C_VEL
LIN {X 0,Y 150.207,Z 193.771,A -85,B 0,C 180,E1 -23907.364,E2 -23907.364} C_VEL
LIN {X 0,Y 150.23,Z 193.768,A -85,B 0,C 180,E1 -23912.718,E2 -23912.718} C_VEL
LIN {X 0,Y 150.338,Z 193.758,A -85,B 0,C 180,E1 -23919.207,E2 -23919.207} C_VEL
LIN {X 0,Y 150.356,Z 193.752,A -85,B 0,C 180,E1 -23923.712,E2 -23923.712} C_VEL
LIN {X 0,Y 150.646,Z 193.719,A -85,B 0,C 180,E1 -23929.245,E2 -23929.245} C_VEL
LIN {X 0,Y 150.733,Z 193.704,A -85,B 0,C 180,E1 -23931.959,E2 -23931.959} C_VEL
LIN {X 0,Y 151.205,Z 193.643,A -85,B 0,C 180,E1 -23940,E2 -23940} C_VEL
LIN {X 0,Y 150.732,Z 193.704,A -85,B 0,C 180,E1 -23948.041,E2 -23948.041} C_VEL
LIN {X 0,Y 150.602,Z 193.724,A -85,B 0,C 180,E1 -23951.507,E2 -23951.507} C_VEL
LIN {X 0,Y 150.355,Z 193.752,A -85,B 0,C 180,E1 -23956.287,E2 -23956.287} C_VEL
LIN {X 0,Y 150.338,Z 193.758,A -85,B 0,C 180,E1 -23960.792,E2 -23960.792} C_VEL
LIN {X 0,Y 150.227,Z 193.768,A -85,B 0,C 180,E1 -23967.28,E2 -23967.28} C_VEL
LIN {X 0,Y 150.201,Z 193.772,A -85,B 0,C 180,E1 -23972.632,E2 -23972.632} C_VEL
LIN {X 0,Y 150.202,Z 193.774,A -85,B 0,C 180,E1 -23977.465,E2 -23977.465} C_VEL
LIN {X 0,Y 150.147,Z 193.779,A -85,B 0,C 180,E1 -23981.51,E2 -23981.51} C_VEL
LIN {X 0,Y 150.128,Z 193.783,A -85,B 0,C 180,E1 -23985.403,E2 -23985.403} C_VEL
LIN {X 0,Y 150.144,Z 193.782,A -85,B 0,C 180,E1 -23989.062,E2 -23989.062} C_VEL
LIN {X 0,Y 150.172,Z 193.774,A -85,B 0,C 180,E1 -23992.711,E2 -23992.711} C_VEL
LIN {X 0,Y 150.209,Z 193.773,A -85,B 0,C 180,E1 -23997.371,E2 -23997.371} C_VEL
LIN {X 0,Y 150.24,Z 193.769,A -85,B 0,C 180,E1 -24002.722,E2 -24002.722} C_VEL
LIN {X 0,Y 150.349,Z 193.753,A -85,B 0,C 180,E1 -24009.21,E2 -24009.21} C_VEL
LIN {X 0,Y 150.369,Z 193.753,A -85,B 0,C 180,E1 -24013.719,E2 -24013.719} C_VEL
LIN {X 0,Y 150.662,Z 193.715,A -85,B 0,C 180,E1 -24019.251,E2 -24019.251} C_VEL
LIN {X 0,Y 150.756,Z 193.707,A -85,B 0,C 180,E1 -24021.965,E2 -24021.965} C_VEL
LIN {X 0,Y 151.208,Z 193.651,A -85,B 0,C 180,E1 -24030.004,E2 -24030.004} C_VEL
LIN {X 0,Y 150.759,Z 193.706,A -85,B 0,C 180,E1 -24038.043,E2 -24038.043} C_VEL
LIN {X 0,Y 150.617,Z 193.72,A -85,B 0,C 180,E1 -24041.511,E2 -24041.511} C_VEL
LIN {X 0,Y 150.365,Z 193.754,A -85,B 0,C 180,E1 -24046.291,E2 -24046.291} C_VEL
LIN {X 0,Y 150.351,Z 193.753,A -85,B 0,C 180,E1 -24050.791,E2 -24050.791} C_VEL
LIN {X 0,Y 150.189,Z 193.776,A -85,B 0,C 180,E1 -24057.241,E2 -24057.241} C_VEL
LIN {X 0,Y 150.214,Z 193.772,A -85,B 0,C 180,E1 -24062.631,E2 -24062.631} C_VEL
LIN {X 0,Y 150.175,Z 193.774,A -85,B 0,C 180,E1 -24067.478,E2 -24067.478} C_VEL
LIN {X 0,Y 150.139,Z 193.782,A -85,B 0,C 180,E1 -24071.5,E2 -24071.5} C_VEL
LIN {X 0,Y 150.133,Z 193.78,A -85,B 0,C 180,E1 -24075.398,E2 -24075.398} C_VEL
LIN {X 0,Y 150.187,Z 193.775,A -85,B 0,C 180,E1 -24079.071,E2 -24079.071} C_VEL
LIN {X 0,Y 150.812,Z 193.698,A -85,B 0,C 180,E1 -24085.999,E2 -24085.999} C_VEL
LIN {X 0,Y 150.885,Z 194.312,A -85,B 0,C 180,E1 -24086.98,E2 -24086.98} C_VEL
LIN {X 0,Y 150.84,Z 196.417,A -85,B 0,C 180,E1 -24089.169,E2 -24089.169} C_VEL
LIN {X 0,Y 149.656,Z 202.096,A -85,B 0,C 180,E1 -24094.998,E2 -24094.998} C_VEL
LIN {X 0,Y 148.76,Z 207.801,A -85,B 0,C 180,E1 -24100.898,E2 -24100.898} C_VEL
LIN {X 0,Y 149.298,Z 217.924,A -85,B 0,C 180,E1 -24111.342,E2 -24111.342} C_VEL
LIN {X 0,Y 150.341,Z 230.17,A -85,B 0,C 180,E1 -24113.289,E2 -24113.289} C_VEL
LIN {X 0,Y 150.662,Z 235.427,A -85,B 0,C 180,E1 -24114.311,E2 -24114.311} C_VEL
LIN {X 0,Y 150.37,Z 245.12,A -85,B 0,C 180,E1 -24116.651,E2 -24116.651} C_VEL
LIN {X 0,Y 150.262,Z 254.216,A -85,B 0,C 180,E1 -24119.33,E2 -24119.33} C_VEL
LIN {X 0,Y 149.984,Z 263.3,A -85,B 0,C 180,E1 -24122.686,E2 -24122.686} C_VEL
LIN {X 0,Y 150.277,Z 272.153,A -85,B 0,C 180,E1 -24126.714,E2 -24126.714} C_VEL
LIN {X 0,Y 151.458,Z 279.335,A -85,B 0,C 180,E1 -24130.697,E2 -24130.697} C_VEL
LIN {X 0,Y 153.287,Z 285.089,A -85,B 0,C 180,E1 -24134.606,E2 -24134.606} C_VEL
LIN {X 0,Y 156.133,Z 289.716,A -85,B 0,C 180,E1 -24138.367,E2 -24138.367} C_VEL
LIN {X 0,Y 160.034,Z 293.3,A -85,B 0,C 180,E1 -24141.918,E2 -24141.918} C_VEL
LIN {X 0,Y 164.662,Z 295.894,A -85,B 0,C 180,E1 -24145.266,E2 -24145.266} C_VEL
LIN {X 0,Y 168.266,Z 297.114,A -85,B 0,C 180,E1 -24147.351,E2 -24147.351} C_VEL
LIN {X 0,Y 176.448,Z 298.251,A -85,B 0,C 180,E1 -24151.185,E2 -24151.185} C_VEL
LIN {X 0,Y 180.951,Z 298.172,A -85,B 0,C 180,E1 -24152.939,E2 -24152.939} C_VEL
LIN {X 0,Y 185.425,Z 297.744,A -85,B 0,C 180,E1 -24154.648,E2 -24154.648} C_VEL
LIN {X 0,Y 188.597,Z 297.319,A -85,B 0,C 180,E1 -24156.601,E2 -24156.601} C_VEL
LIN {X 0,Y 191.417,Z 296.851,A -85,B 0,C 180,E1 -24158.621,E2 -24158.621} C_VEL
LIN {X 0,Y 192.884,Z 296.64,A -85,B 0,C 180,E1 -24160.074,E2 -24160.074} C_VEL
LIN {X 0,Y 194.593,Z 296.779,A -85,B 0,C 180,E1 -24163.331,E2 -24163.331} C_VEL
LIN {X 0,Y 194.802,Z 297.541,A -85,B 0,C 180,E1 -24166.183,E2 -24166.183} C_VEL
LIN {X 0,Y 194.451,Z 297.793,A -85,B 0,C 180,E1 -24166.626,E2 -24166.626} C_VEL
LIN {X 0,Y 184.024,Z 301.335,A -85,B 0,C 180,E1 -24169.802,E2 -24169.802} C_VEL
LIN {X 0,Y 175.468,Z 303.309,A -85,B 0,C 180,E1 -24173.069,E2 -24173.069} C_VEL
LIN {X 0,Y 167.486,Z 304.183,A -85,B 0,C 180,E1 -24176.937,E2 -24176.937} C_VEL
LIN {X 0,Y 161.134,Z 303.961,A -85,B 0,C 180,E1 -24181.325,E2 -24181.325} C_VEL
LIN {X 0,Y 156.032,Z 302.587,A -85,B 0,C 180,E1 -24186.081,E2 -24186.081} C_VEL
LIN {X 0,Y 152.545,Z 300.065,A -85,B 0,C 180,E1 -24191.182,E2 -24191.182} C_VEL
LIN {X 0,Y 150.834,Z 296.406,A -85,B 0,C 180,E1 -24196.524,E2 -24196.524} C_VEL
LIN {X 0,Y 150.755,Z 291.387,A -85,B 0,C 180,E1 -24201.956,E2 -24201.956} C_VEL
LIN {X 0,Y 151.573,Z 286.534,A -85,B 0,C 180,E1 -24206.008,E2 -24206.008} C_VEL
LIN {X 0,Y 152.07,Z 283.612,A -85,B 0,C 180,E1 -24208.009,E2 -24208.009} C_VEL
LIN {X 0,Y 152.131,Z 278.771,A -85,B 0,C 180,E1 -24210.658,E2 -24210.658} C_VEL
LIN {X 0,Y 152.076,Z 272.869,A -85,B 0,C 180,E1 -24213.307,E2 -24213.307} C_VEL
LIN {X 0,Y 152.004,Z 262.769,A -85,B 0,C 180,E1 -24216.967,E2 -24216.967} C_VEL
LIN {X 0,Y 152.223,Z 252.258,A -85,B 0,C 180,E1 -24219.966,E2 -24219.966} C_VEL
LIN {X 0,Y 152.477,Z 243.545,A -85,B 0,C 180,E1 -24221.966,E2 -24221.966} C_VEL
LIN {X 0,Y 151.061,Z 231.428,A -85,B 0,C 180,E1 -24223.961,E2 -24223.961} C_VEL
LIN {X 0,Y 150.327,Z 219.645,A -85,B 0,C 180,E1 -24225.503,E2 -24225.503} C_VEL
LIN {X 0,Y 149.695,Z 215.556,A -85,B 0,C 180,E1 -24229.182,E2 -24229.182} C_VEL
LIN {X 0,Y 152.128,Z 205.101,A -85,B 0,C 180,E1 -24238.626,E2 -24238.626} C_VEL
LIN {X 0,Y 152.722,Z 203.081,A -85,B 0,C 180,E1 -24240.406,E2 -24240.406} C_VEL
LIN {X 0,Y 151.314,Z 197.452,A -85,B 0,C 180,E1 -24245.486,E2 -24245.486} C_VEL
LIN {X 0,Y 151.08,Z 196.407,A -85,B 0,C 180,E1 -24246.448,E2 -24246.448} C_VEL
LIN {X 0,Y 150.489,Z 195.223,A -85,B 0,C 180,E1 -24247.84,E2 -24247.84} C_VEL
LIN {X 0,Y 148.849,Z 194.353,A -85,B 0,C 180,E1 -24249.979,E2 -24249.979} C_VEL
LIN {X 0,Y 145.451,Z 194.366,A -85,B 0,C 180,E1 -24253.647,E2 -24253.647} C_VEL
LIN {X 0,Y 143.184,Z 194.644,A -85,B 0,C 180,E1 -24257.566,E2 -24257.566} C_VEL
LIN {X 0,Y 143.082,Z 194.653,A -85,B 0,C 180,E1 -24258.376,E2 -24258.376} C_VEL
LIN {X 0,Y 143.113,Z 194.657,A -85,B 0,C 180,E1 -24263.893,E2 -24263.893} C_VEL
LIN {X 0,Y 143.175,Z 194.647,A -85,B 0,C 180,E1 -24267.319,E2 -24267.319} C_VEL
LIN {X 0,Y 143.178,Z 194.648,A -85,B 0,C 180,E1 -24272.062,E2 -24272.062} C_VEL
LIN {X 0,Y 143.264,Z 194.639,A -85,B 0,C 180,E1 -24278.745,E2 -24278.745} C_VEL
LIN {X 0,Y 143.293,Z 194.629,A -85,B 0,C 180,E1 -24282.885,E2 -24282.885} C_VEL
LIN {X 0,Y 143.583,Z 194.599,A -85,B 0,C 180,E1 -24288.709,E2 -24288.709} C_VEL
LIN {X 0,Y 143.653,Z 194.585,A -85,B 0,C 180,E1 -24291.56,E2 -24291.56} C_VEL
LIN {X 0,Y 144.164,Z 194.52,A -85,B 0,C 180,E1 -24300,E2 -24300} C_VEL
LIN {X 0,Y 143.653,Z 194.586,A -85,B 0,C 180,E1 -24308.44,E2 -24308.44} C_VEL
LIN {X 0,Y 143.536,Z 194.604,A -85,B 0,C 180,E1 -24311.713,E2 -24311.713} C_VEL
LIN {X 0,Y 143.293,Z 194.629,A -85,B 0,C 180,E1 -24317.114,E2 -24317.114} C_VEL
LIN {X 0,Y 143.263,Z 194.639,A -85,B 0,C 180,E1 -24321.254,E2 -24321.254} C_VEL
LIN {X 0,Y 143.171,Z 194.649,A -85,B 0,C 180,E1 -24327.933,E2 -24327.933} C_VEL
LIN {X 0,Y 143.153,Z 194.649,A -85,B 0,C 180,E1 -24333.435,E2 -24333.435} C_VEL
LIN {X 0,Y 143.067,Z 194.664,A -85,B 0,C 180,E1 -24339.688,E2 -24339.688} C_VEL
LIN {X 0,Y 143.058,Z 194.66,A -85,B 0,C 180,E1 -24343.454,E2 -24343.454} C_VEL
LIN {X 0,Y 143.06,Z 194.666,A -85,B 0,C 180,E1 -24347.467,E2 -24347.467} C_VEL
LIN {X 0,Y 143.07,Z 194.658,A -85,B 0,C 180,E1 -24351.81,E2 -24351.81} C_VEL
LIN {X 0,Y 143.176,Z 194.649,A -85,B 0,C 180,E1 -24357.326,E2 -24357.326} C_VEL
LIN {X 0,Y 143.186,Z 194.646,A -85,B 0,C 180,E1 -24362.067,E2 -24362.067} C_VEL
LIN {X 0,Y 143.275,Z 194.633,A -85,B 0,C 180,E1 -24368.749,E2 -24368.749} C_VEL
LIN {X 0,Y 143.307,Z 194.634,A -85,B 0,C 180,E1 -24372.892,E2 -24372.892} C_VEL
LIN {X 0,Y 143.593,Z 194.596,A -85,B 0,C 180,E1 -24378.715,E2 -24378.715} C_VEL
LIN {X 0,Y 143.675,Z 194.588,A -85,B 0,C 180,E1 -24381.566,E2 -24381.566} C_VEL
LIN {X 0,Y 144.169,Z 194.528,A -85,B 0,C 180,E1 -24390.004,E2 -24390.004} C_VEL
LIN {X 0,Y 143.677,Z 194.587,A -85,B 0,C 180,E1 -24398.443,E2 -24398.443} C_VEL
LIN {X 0,Y 143.551,Z 194.599,A -85,B 0,C 180,E1 -24401.717,E2 -24401.717} C_VEL
LIN {X 0,Y 143.303,Z 194.635,A -85,B 0,C 180,E1 -24407.117,E2 -24407.117} C_VEL
LIN {X 0,Y 143.275,Z 194.633,A -85,B 0,C 180,E1 -24411.252,E2 -24411.252} C_VEL
LIN {X 0,Y 143.147,Z 194.651,A -85,B 0,C 180,E1 -24417.904,E2 -24417.904} C_VEL
LIN {X 0,Y 143.144,Z 194.654,A -85,B 0,C 180,E1 -24423.42,E2 -24423.42} C_VEL
LIN {X 0,Y 143.058,Z 194.661,A -85,B 0,C 180,E1 -24429.696,E2 -24429.696} C_VEL
LIN {X 0,Y 143.04,Z 194.666,A -85,B 0,C 180,E1 -24433.467,E2 -24433.467} C_VEL
LIN {X 0,Y 143.084,Z 194.655,A -85,B 0,C 180,E1 -24437.463,E2 -24437.463} C_VEL
LIN {X 0,Y 143.469,Z 194.612,A -85,B 0,C 180,E1 -24443.997,E2 -24443.997} C_VEL
LIN {X 0,Y 143.812,Z 194.655,A -85,B 0,C 180,E1 -24446.842,E2 -24446.842} C_VEL
LIN {X 0,Y 143.735,Z 196.73,A -85,B 0,C 180,E1 -24449.109,E2 -24449.109} C_VEL
LIN {X 0,Y 142.494,Z 202.405,A -85,B 0,C 180,E1 -24455.214,E2 -24455.214} C_VEL
LIN {X 0,Y 141.61,Z 208.235,A -85,B 0,C 180,E1 -24461.552,E2 -24461.552} C_VEL
LIN {X 0,Y 142.28,Z 217.668,A -85,B 0,C 180,E1 -24471.759,E2 -24471.759} C_VEL
LIN {X 0,Y 142.482,Z 218.043,A -85,B 0,C 180,E1 -24472.15,E2 -24472.15} C_VEL
LIN {X 0,Y 143.772,Z 231.49,A -85,B 0,C 180,E1 -24474.39,E2 -24474.39} C_VEL
LIN {X 0,Y 143.755,Z 240.717,A -85,B 0,C 180,E1 -24476.497,E2 -24476.497} C_VEL
LIN {X 0,Y 143.552,Z 251.595,A -85,B 0,C 180,E1 -24479.65,E2 -24479.65} C_VEL
LIN {X 0,Y 143.309,Z 261.988,A -85,B 0,C 180,E1 -24483.515,E2 -24483.515} C_VEL
LIN {X 0,Y 143.688,Z 271.058,A -85,B 0,C 180,E1 -24487.73,E2 -24487.73} C_VEL
LIN {X 0,Y 145.012,Z 278.43,A -85,B 0,C 180,E1 -24491.887,E2 -24491.887} C_VEL
LIN {X 0,Y 147.463,Z 285.248,A -85,B 0,C 180,E1 -24496.616,E2 -24496.616} C_VEL
LIN {X 0,Y 150.762,Z 289.935,A -85,B 0,C 180,E1 -24500.465,E2 -24500.465} C_VEL
LIN {X 0,Y 155.006,Z 293.577,A -85,B 0,C 180,E1 -24504.083,E2 -24504.083} C_VEL
LIN {X 0,Y 158.281,Z 295.458,A -85,B 0,C 180,E1 -24506.361,E2 -24506.361} C_VEL
LIN {X 0,Y 161.974,Z 296.954,A -85,B 0,C 180,E1 -24508.509,E2 -24508.509} C_VEL
LIN {X 0,Y 170.39,Z 298.678,A -85,B 0,C 180,E1 -24512.426,E2 -24512.426} C_VEL
LIN {X 0,Y 175.031,Z 298.905,A -85,B 0,C 180,E1 -24514.204,E2 -24514.204} C_VEL
LIN {X 0,Y 179.646,Z 298.773,A -85,B 0,C 180,E1 -24515.932,E2 -24515.932} C_VEL
LIN {X 0,Y 182.876,Z 298.613,A -85,B 0,C 180,E1 -24517.944,E2 -24517.944} C_VEL
LIN {X 0,Y 185.656,Z 298.429,A -85,B 0,C 180,E1 -24520.056,E2 -24520.056} C_VEL
LIN {X 0,Y 186.596,Z 298.441,A -85,B 0,C 180,E1 -24521.12,E2 -24521.12} C_VEL
LIN {X 0,Y 187.231,Z 298.583,A -85,B 0,C 180,E1 -24522.505,E2 -24522.505} C_VEL
LIN {X 0,Y 187.878,Z 299.126,A -85,B 0,C 180,E1 -24525.295,E2 -24525.295} C_VEL
LIN {X 0,Y 184.19,Z 300.278,A -85,B 0,C 180,E1 -24526.618,E2 -24526.618} C_VEL
LIN {X 0,Y 174.39,Z 302.483,A -85,B 0,C 180,E1 -24529.845,E2 -24529.845} C_VEL
LIN {X 0,Y 165.596,Z 303.439,A -85,B 0,C 180,E1 -24533.542,E2 -24533.542} C_VEL
LIN {X 0,Y 158.095,Z 303.27,A -85,B 0,C 180,E1 -24537.757,E2 -24537.757} C_VEL
LIN {X 0,Y 152.162,Z 302.06,A -85,B 0,C 180,E1 -24542.487,E2 -24542.487} C_VEL
LIN {X 0,Y 147.661,Z 299.71,A -85,B 0,C 180,E1 -24547.615,E2 -24547.615} C_VEL
LIN {X 0,Y 144.95,Z 296.249,A -85,B 0,C 180,E1 -24553.083,E2 -24553.083} C_VEL
LIN {X 0,Y 144.073,Z 291.597,A -85,B 0,C 180,E1 -24558.744,E2 -24558.744} C_VEL
LIN {X 0,Y 144.517,Z 287.145,A -85,B 0,C 180,E1 -24563.013,E2 -24563.013} C_VEL
LIN {X 0,Y 145.526,Z 281.572,A -85,B 0,C 180,E1 -24567.228,E2 -24567.228} C_VEL
LIN {X 0,Y 145.639,Z 275.198,A -85,B 0,C 180,E1 -24570.687,E2 -24570.687} C_VEL
LIN {X 0,Y 145.399,Z 268.756,A -85,B 0,C 180,E1 -24573.459,E2 -24573.459} C_VEL
LIN {X 0,Y 145.384,Z 258.882,A -85,B 0,C 180,E1 -24576.937,E2 -24576.937} C_VEL
LIN {X 0,Y 145.559,Z 249.019,A -85,B 0,C 180,E1 -24579.725,E2 -24579.725} C_VEL
LIN {X 0,Y 145.593,Z 241.506,A -85,B 0,C 180,E1 -24581.435,E2 -24581.435} C_VEL
LIN {X 0,Y 144.069,Z 228.76,A -85,B 0,C 180,E1 -24583.525,E2 -24583.525} C_VEL
LIN {X 0,Y 143.487,Z 219.683,A -85,B 0,C 180,E1 -24584.715,E2 -24584.715} C_VEL
LIN {X 0,Y 142.625,Z 215.509,A -85,B 0,C 180,E1 -24588.676,E2 -24588.676} C_VEL
LIN {X 0,Y 145.301,Z 204.2,A -85,B 0,C 180,E1 -24599.467,E2 -24599.467} C_VEL
LIN {X 0,Y 145.558,Z 203.016,A -85,B 0,C 180,E1 -24600.568,E2 -24600.568} C_VEL
LIN {X 0,Y 143.876,Z 196.164,A -85,B 0,C 180,E1 -24607.11,E2 -24607.11} C_VEL
LIN {X 0,Y 143.515,Z 194.604,A -85,B 0,C 180,E1 -24608.741,E2 -24608.741} C_VEL
LIN {X 0,Y 143.157,Z 194.652,A -85,B 0,C 180,E1 -24613.41,E2 -24613.41} C_VEL
LIN {X 0,Y 143.082,Z 194.653,A -85,B 0,C 180,E1 -24618.376,E2 -24618.376} C_VEL
LIN {X 0,Y 142.729,Z 194.705,A -85,B 0,C 180,E1 -24619.946,E2 -24619.946} C_VEL
LIN {X 0,Y 141.347,Z 194.879,A -85,B 0,C 180,E1 -24622.271,E2 -24622.271} C_VEL
LIN {X 0,Y 136.304,Z 195.506,A -85,B 0,C 180,E1 -24629.424,E2 -24629.424} C_VEL
LIN {X 0,Y 136.072,Z 195.533,A -85,B 0,C 180,E1 -24631.108,E2 -24631.108} C_VEL
